# B&R Automation Studio project PLC code - cp (part 6)

#### HeightTracking.st
```iecst
ACTION RunHeightArray:

	// ------------------------------------------------------------------
	// Matrix advance and calculate the maximum

	//Move the values of the array
	ShiftArrayForward(ADR(iHeightArray), SIZEOF(iHeightArray), SIZEOF(iHeightArray[0]), iPositionsToRunArray, iTotalBlocksLengh);

	// High Ctrl data to Matrix
	// Loading data from sensors to
	IF gPhotoCells.status.xInstalled THEN
		LoadHeightFromArraySensor;
	END_IF
	IF gDing.State.xDingInstalled OR gBasicDetectMedia.Status.xInstalled THEN
		LoadHeightFromAnalogSensor;
	END_IF

	// Analyze height data and assign maximum height per section
	ResetMaxHeigh;
	FOR iIndexArray:= iTotalBlocksLengh TO iPositionsToRunArray BY -1 DO
		//Update te value of the thickness in the matrix
		AssignMaxHeighIndex;
	END_FOR

END_ACTION

ACTION ResetMaxHeigh:

	// It allows changes on height block correction when It changes Hand Printer
	FOR iIndexSection:=1 TO iTotalSections DO
		iMaxHeigh[iIndexSection]:=0;
	END_FOR

END_ACTION

ACTION AssignMaxHeighIndex:

	//Calculate the maximum of each section
	FOR iIndexSection:=1 TO iTotalSections DO
		//If the section is not enabled, do not calculate any Max
		IF dataHeigh.parameters.sections[iIndexSection].xEnabled THEN

			//If the Section does not correspond with the Index in Matrix, do not calculate Max
			IF iIndexArray > dataHeigh.parameters.sections[iIndexSection].iStart AND
				iIndexArray <= dataHeigh.parameters.sections[iIndexSection].iEnd 	 THEN

				iMaxHeigh[iIndexSection]:= MAX(iHeightArray[iIndexArray], iMaxHeigh[iIndexSection]);
			END_IF
		END_IF

	END_FOR

END_ACTION

ACTION AssignMaxHeight:

	//Calculate the maximum of each section
	FOR iIndexSection:=1 TO iTotalSections DO
		//If the section is not enabled, do not calculate any Max
		IF dataHeigh.parameters.sections[iIndexSection].xEnabled THEN
			FOR iIndexArray:= dataHeigh.parameters.sections[iIndexSection].iStart TO dataHeigh.parameters.sections[iIndexSection].iEnd DO
				iMaxHeigh[iIndexSection]:= MAX(iHeightArray[iIndexArray], iMaxHeigh[iIndexSection]);
			END_FOR
		END_IF
	END_FOR

END_ACTION

ACTION LoadHeightFromAnalogSensor:
	//TODO. convert in a FUNCTION to use 3 times

	// Fill-in moved spaces with new data
	iCurrentMediaHeight := 0;
	IF dataHeigh.Internal.iFastValues >= iPositionsToRunArray THEN
		// More values than holes to fill-in. Distribution of data
		rValuesPerPosition :=  dataHeigh.Internal.rFastValues / UINT_TO_REAL(iPositionsToRunArray);
		FOR iIndexArray:=0 TO iPositionsToRunArray -1 DO
			iHeightArray[iIndexArray + iAnalogSensorPosition] := 0;
			FOR iIndexNewMediaArray := INT_TO_UINT( TRUNC(UINT_TO_REAL(iIndexArray) * rValuesPerPosition )) TO INT_TO_UINT(TRUNC(UINT_TO_REAL(iIndexArray) * rValuesPerPosition )) DO
				iHeightArray[iIndexArray + iAnalogSensorPosition] := MAX(iHeightArray[iIndexArray + iAnalogSensorPosition], dataHeigh.Internal.AnalogHeightValues[iIndexNewMediaArray]);
				iCurrentMediaHeight := MAX(iCurrentMediaHeight, dataHeigh.Internal.AnalogHeightValues[iIndexNewMediaArray]);
			END_FOR
		END_FOR
	ELSE
		// More holes than data. Ampliation of data
		rValuesPerPosition :=  UINT_TO_REAL(iPositionsToRunArray) / dataHeigh.Internal.rFastValues;
		FOR iIndexNewMediaArray:=0 TO REAL_TO_UINT(dataHeigh.Internal.rFastValues) -1 DO
			FOR iIndexArray := INT_TO_UINT(TRUNC(UINT_TO_REAL(iIndexNewMediaArray) * rValuesPerPosition )) TO INT_TO_UINT(TRUNC(UINT_TO_REAL(iIndexNewMediaArray) * rValuesPerPosition )) DO
				iHeightArray[iIndexArray + iAnalogSensorPosition] :=dataHeigh.Internal.AnalogHeightValues[iIndexNewMediaArray];
				iCurrentMediaHeight := MAX(iCurrentMediaHeight, dataHeigh.Internal.AnalogHeightValues[iIndexNewMediaArray]);
			END_FOR
		END_FOR
	END_IF
	gThicknessCtrl.status.Heigh.iMediaHeigh := iCurrentMediaHeight;

END_ACTION

ACTION LoadHeightFromArraySensor:
	//TODO. convert in a FUNCTION to use 3 times

	// Fill-in moved spaces with new data
	iCurrentMediaHeight := 0;
	IF dataHeigh.Internal.iFastValues >= iPositionsToRunArray THEN
		// More values than holes to fill-in. Distribution of data
		rValuesPerPosition :=  dataHeigh.Internal.rFastValues / UINT_TO_REAL(iPositionsToRunArray);
		FOR iIndexArray:=0 TO iPositionsToRunArray -1 DO
			iHeightArray[iIndexArray + iArraySensorPosition] := 0;
			FOR iIndexNewMediaArray := INT_TO_UINT(TRUNC(UINT_TO_REAL(iIndexArray) * rValuesPerPosition )) TO INT_TO_UINT(TRUNC(UINT_TO_REAL(iIndexArray) * rValuesPerPosition )) DO
				iHeightArray[iIndexArray + iArraySensorPosition] := MAX(iHeightArray[iIndexArray + iArraySensorPosition], dataHeigh.Internal.ArrayHeightValues[iIndexNewMediaArray]);
				iCurrentMediaHeight := MAX(iCurrentMediaHeight, dataHeigh.Internal.ArrayHeightValues[iIndexNewMediaArray]);
			END_FOR
		END_FOR
	ELSE
		// More holes than data. Ampliation of data
		rValuesPerPosition :=  UINT_TO_REAL(iPositionsToRunArray) / dataHeigh.Internal.rFastValues;
		FOR iIndexNewMediaArray:=0 TO REAL_TO_UINT(dataHeigh.Internal.rFastValues) -1 DO
			FOR iIndexArray := INT_TO_UINT(TRUNC(UINT_TO_REAL(iIndexNewMediaArray) * rValuesPerPosition )) TO INT_TO_UINT(TRUNC(UINT_TO_REAL(iIndexNewMediaArray) * rValuesPerPosition )) DO
				iHeightArray[iIndexArray + iArraySensorPosition] :=dataHeigh.Internal.ArrayHeightValues[iIndexNewMediaArray];
				iCurrentMediaHeight := MAX(iCurrentMediaHeight, dataHeigh.Internal.ArrayHeightValues[iIndexNewMediaArray]);
			END_FOR
		END_FOR
	END_IF
	gThicknessCtrl.status.Heigh.iMediaHeigh := iCurrentMediaHeight;

END_ACTION
```

#### MediaTrackingFunct.st
```iecst
ACTION MoveMediaFromNewToInsideL1:

	IF MediaTracking_iTotalInsideL1 = THICK_MEDIATRACKING_MAX_MEDIA THEN
		// TODO: Raise alarm of received media without free space
		RETURN;
	END_IF

	// Moving from New to Inside
	IF dataHeigh.status.xNewMediaStackEnabled THEN
		// Managing Media and Energy
		MediaTrackingInsideL1[MediaTracking_iTotalInsideL1] := NewMediaStackL1[0];
	ELSE
		// Manage Energy information
		MediaEnergyRackL1[EnergyRack_iIndexL1] := dataHeigh.parameters.ContinuousMedia.Energy;
		MediaTrackingInsideL1[MediaTracking_iTotalInsideL1].iIndexMediaEnergy := EnergyRack_iIndexL1;
		MediaTrackingInsideL1[MediaTracking_iTotalInsideL1].pMediaEnery := ADR(MediaEnergyRackL1[EnergyRack_iIndexL1]);
		EnergyRack_iIndexL1 := EnergyRack_iIndexL1 + 1;
		IF EnergyRack_iIndexL1 > THICK_MEDIATRACKING_MAX_MEDIA_x2 THEN
			EnergyRack_iIndexL1 := 0;
		END_IF
		// Managing media
		MediaTrackingInsideL1[MediaTracking_iTotalInsideL1].Media := dataHeigh.parameters.ContinuousMedia.MediaData;
	END_IF

	MediaTrackingInsideL1[MediaTracking_iTotalInsideL1].HeadPosition := iIndexEnteringMedia;
	MediaTracking_iTotalInsideL1 := MediaTracking_iTotalInsideL1 + 1;
	AssignEnteringMediaL1;

	// Removing from New overwriting the array
	IF dataHeigh.status.xNewMediaStackEnabled THEN
		ShiftArrayBackward(ADR(NewMediaStackL1), SIZEOF(NewMediaStackL1), SIZEOF(NewMediaStackL1[0]), 1, Stack_iTotalNewMediaL1);
		Stack_iTotalNewMediaL1 := UINT_SUB(Stack_iTotalNewMediaL1, 1);
	END_IF

	AddMediaTrackingEvents(diTotalCmBelt, HEAD_DETECTED, ADR(TrackingEventsArray));

END_ACTION

ACTION MoveMediaFromNewToInsideL2:

	IF MediaTracking_iTotalInsideL2 = THICK_MEDIATRACKING_MAX_MEDIA THEN
		// TODO: Raise alarm of received media without free space
		RETURN;
	END_IF

	// Moving from New to Inside
	IF dataHeigh.status.xNewMediaStackEnabled THEN
		// Managing Media and Energy
		MediaTrackingInsideL2[MediaTracking_iTotalInsideL2] := NewMediaStackL2[0];
	ELSE
		// Manage Energy information
		MediaEnergyRackL2[EnergyRack_iIndexL2] := dataHeigh.parameters.ContinuousMedia.Energy;
		MediaTrackingInsideL2[MediaTracking_iTotalInsideL2].iIndexMediaEnergy := EnergyRack_iIndexL2;
		MediaTrackingInsideL2[MediaTracking_iTotalInsideL2].pMediaEnery := ADR(MediaEnergyRackL2[EnergyRack_iIndexL2]);
		EnergyRack_iIndexL2 := EnergyRack_iIndexL2 + 1;
		IF EnergyRack_iIndexL2 > THICK_MEDIATRACKING_MAX_MEDIA_x2 THEN
			EnergyRack_iIndexL2 := 0;
		END_IF
		// Managing media
		MediaTrackingInsideL2[MediaTracking_iTotalInsideL2].Media := dataHeigh.parameters.ContinuousMedia.MediaData;
	END_IF

	MediaTrackingInsideL2[MediaTracking_iTotalInsideL2].HeadPosition := iIndexEnteringMedia;
	MediaTracking_iTotalInsideL2 := MediaTracking_iTotalInsideL2 + 1;
	AssignEnteringMediaL2;

	// Removing from New overwriting the array
	IF dataHeigh.status.xNewMediaStackEnabled THEN
		ShiftArrayBackward(ADR(NewMediaStackL2), SIZEOF(NewMediaStackL2), SIZEOF(NewMediaStackL2[0]), 1, Stack_iTotalNewMediaL2);
		Stack_iTotalNewMediaL2 := UINT_SUB(Stack_iTotalNewMediaL2, 1);
	END_IF

	AddMediaTrackingEvents(diTotalCmBelt, HEAD_DETECTED, ADR(TrackingEventsArray));

END_ACTION

ACTION MoveMediaFromInsideToOutL1:

	// Removing from New overwriting the array
	ShiftArrayBackward(ADR(MediaTrackingInsideL1), SIZEOF(MediaTrackingInsideL1), SIZEOF(MediaTrackingInsideL1[0]), 1, MediaTracking_iTotalInsideL1);
	MediaTracking_iTotalInsideL1 := UINT_SUB(MediaTracking_iTotalInsideL1, 1);
	AssignEnteringMediaL1;
	xExitingMediaL1 := TRUE;

END_ACTION

ACTION MoveMediaFromInsideToOutL2:

	// Removing from New overwriting the array
	ShiftArrayBackward(ADR(MediaTrackingInsideL2), SIZEOF(MediaTrackingInsideL2), SIZEOF(MediaTrackingInsideL2[0]), 1, MediaTracking_iTotalInsideL2);
	MediaTracking_iTotalInsideL2 := UINT_SUB(MediaTracking_iTotalInsideL2, 1);
	AssignEnteringMediaL2;
	xExitingMediaL2 := TRUE;

END_ACTION

ACTION AssignEnteringMediaL1:

	// Need to protect the case when exiting one media and no other media inside. In this case pointing to an empty location, but no errors
	IF MediaTracking_iTotalInsideL1 > 0 THEN
		EnteringMediaL1 ACCESS ADR(MediaTrackingInsideL1[MediaTracking_iTotalInsideL1-1].Media);
	ELSE
		EnteringMediaL1 ACCESS ADR(MediaTrackingInsideL1[0].Media);
	END_IF

END_ACTION

ACTION AssignEnteringMediaL2:

	// Need to protect the case when exiting one media and no other media inside. In this case pointing to an empty location, but no errors
	IF MediaTracking_iTotalInsideL2 > 0 THEN
		EnteringMediaL2 ACCESS ADR(MediaTrackingInsideL2[MediaTracking_iTotalInsideL2-1].Media);
	ELSE
		EnteringMediaL2 ACCESS ADR(MediaTrackingInsideL2[0].Media);
	END_IF

END_ACTION

ACTION RunMediaInsidePositions:

	RunMediaInsidePositionsL1;
	IF dataHeigh.parameters.xDoubleLine THEN
		RunMediaInsidePositionsL2;
	END_IF

END_ACTION

ACTION RunMediaInsidePositionsL1:

	IF MediaTracking_iTotalInsideL1 = 0 THEN
		RETURN;
	END_IF

	FOR iIndexArray := 0 TO MediaTracking_iTotalInsideL1 -1 DO
		MediaTrackingInsideL1[iIndexArray].HeadPosition := MediaTrackingInsideL1[iIndexArray].HeadPosition + iPositionsToRunArray;
		// If tail position is <>0 is because it has been asigned
		IF MediaTrackingInsideL1[iIndexArray].TailPosition <> 0 THEN
			MediaTrackingInsideL1[iIndexArray].TailPosition := MediaTrackingInsideL1[iIndexArray].TailPosition + iPositionsToRunArray;
		END_IF
	END_FOR

END_ACTION

ACTION RunMediaInsidePositionsL2:

	IF MediaTracking_iTotalInsideL2 = 0 THEN
		RETURN;
	END_IF

	FOR iIndexArray := 0 TO MediaTracking_iTotalInsideL2 -1 DO
		MediaTrackingInsideL2[iIndexArray].HeadPosition := MediaTrackingInsideL2[iIndexArray].HeadPosition + iPositionsToRunArray;
		// If tail position is <>0 is because it has been asigned
		IF MediaTrackingInsideL2[iIndexArray].TailPosition <> 0 THEN
			MediaTrackingInsideL2[iIndexArray].TailPosition := MediaTrackingInsideL2[iIndexArray].TailPosition + iPositionsToRunArray;
		END_IF
	END_FOR

END_ACTION
```

#### RejectTracking.st
```iecst
ACTION RunRejectArray:

	//Need to run the matrix through all belts
	ShiftArrayForward(ADR(ValidMedia), SIZEOF(ValidMedia), SIZEOF(ValidMedia[0]), iPositionsToRunArray, iMaxTrackingPosition + 5);

	// To Clarify if Command for 1 or Order for all till contrary order
	IF EDGEPOS(dataHeigh.Commands.xRushProof) THEN
		xRushProof:=TRUE;
		iRushProofCounter := iRushProofCounter + 1; //To be shown on UI. Useful for users and debugging
		LogRushProof;

		MarkBoardAsRejectedToTheFrontEdge;
	END_IF

	// When receiving the signal of media detected to Reject, run the matrix and mark all boards as ToReject
	// This will ocurr the next scan cycle of the detection, but it is no a problem in this case
	IF EDGENEG(dataHeigh.parameters.xBlockInProperPrintingPosition) OR dataHeigh.status.Detection.xMediaToRejectDetected THEN
		IF gMachine.St.AutoMode.xProduction THEN
			MarkAllBoardsBelowMachineAsRejected;
		END_IF
		xReturningFromReject := TRUE;
	END_IF

	//To write the matrix
	IF dataHeigh.parameters.xBlockInProperPrintingPosition AND NOT dataHeigh.Orders.xDiscardAllMedia THEN
		IF NOT xRushProof THEN

			IF NOT xReturningFromReject THEN
				// This is the standard behaviour. MOST OF TIMES THROUGH HERE
				iNewValidMedia := MEDIATRACKING_VALID;
				LoadNewValidMediaData;
			ELSE
				//   This is the behaviourr while finishing the Reject state,
				// and searching for a gap in the media entering to considering finished
				IF dataHeigh.parameters.Detection.ProductDetect.xFixedSensor THEN
					iNewValidMedia := MEDIATRACKING_INVALID;
				ELSE
					iNewValidMedia := MEDIATRACKING_UNKNOWN;
				END_IF
				LoadNewValidMediaData;
				DetectGapEnteringTheMachine;
			END_IF
		ELSE
			// Review Rear Edge. Invalid if not Edge. Valid after the edge
			CheckRearEdgeofRejectedBoard;
		END_IF
	ELSE
		IF dataHeigh.parameters.Detection.ProductDetect.xFixedSensor THEN
			iNewValidMedia := MEDIATRACKING_INVALID;
		ELSE
			iNewValidMedia := MEDIATRACKING_UNKNOWN;
		END_IF
		LoadNewValidMediaData;

		xRushProof:=FALSE;
	END_IF

	// Just update if the new data is written in the positions moved previously

END_ACTION

ACTION LoadNewValidMediaData:
	FOR iIndexArray := 0 TO iPositionsToRunArray -1 DO
		ValidMedia[iIndexArray + iProductDetectSensorPosition] := iNewValidMedia;
	END_FOR
END_ACTION

ACTION ReviewRejectActivation:

	//[RGP] This part must be located in code executed much faster: less than (MinGap/MaxBeltSpeed)
	//We need TO force gaps TO be written with a PDsignal filter, TO avoid "iPositionsToRunArray" TO mask them
	//we can check previous index (iRejectLengthAdjustment-X). X: Positions in matrix forced to be 0, as a gap

	FastReviewReject;

	//Overwritting valid media array to mark boards below bars when block raises to safe position
	//[RGP] 15274: Overwritting matrix position to know which boards are below block's bars when empty belt mode.
	IF EDGEPOS(dataHeigh.Orders.xDiscardAllMedia) THEN
		FOR iIndex := dataHeigh.parameters.Detection.ProductDetect.iSensorPosition TO dataHeigh.parameters.iTotalBlocksLengh DO
			IF dataHeigh.parameters.Detection.ProductDetect.xFixedSensor THEN
				ValidMedia[iIndex] := MEDIATRACKING_INVALID;
			ELSE
				ValidMedia[iIndex] := MEDIATRACKING_UNKNOWN;
			END_IF
		END_FOR
	END_IF

	ton_PhysicalHoldReject(IN:=gMachine.In.Buttons.xReset, PT:=T#2S);
	xHoldReject := ValidMedia[iHoldRejectLengthAdjustment] = MEDIATRACKING_UNKNOWN;

	IF EDGEPOS(xHoldReject) THEN
		AddMediaTrackingEvents(diTotalCmBelt + iHoldRejectLengthAdjustment, START_HOLDREJEC, ADR(TrackingEventsArray));
	END_IF
	IF EDGENEG(xHoldReject) THEN
		AddMediaTrackingEvents(diTotalCmBelt + iHoldRejectLengthAdjustment, END_HOLDREJECT, ADR(TrackingEventsArray));
	END_IF

	// Out signals
	dataHeigh.Outputs.xHoldReject := ton_PhysicalHoldReject.Q OR xHoldReject;

END_ACTION

ACTION MarkBoardAsRejectedToTheFrontEdge:

	// Searching for the gap in xMediaTracking
	FOR iIndex:=iProductDetectSensorPosition TO iMAXTRACKINGARRAY DO
		// Searching for the gap in xMediaTracking to Stop
		IF xMediaTracking[iIndex] = 0  THEN
			EXIT;
		END_IF
		ValidMedia[iIndex] := MEDIATRACKING_INVALID;
	END_FOR

END_ACTION

ACTION DetectGapEnteringTheMachine:

	// Searching for the gap in xMediaTracking
	FOR iIndex:=iProductDetectSensorPosition + iPositionsToRunArray TO iProductDetectSensorPosition BY -1 DO
		// Searching for the gap in xMediaTracking to Stop
		IF xMediaTracking[iIndex] = 0  THEN
			xReturningFromReject := FALSE;
			EXIT;
		END_IF
	END_FOR

END_ACTION

ACTION CheckRearEdgeofRejectedBoard:

	// Searching for the gap in xMediaTracking
	FOR iIndex:=iProductDetectSensorPosition + iPositionsToRunArray TO iProductDetectSensorPosition BY -1 DO

		IF xMediaTracking[iIndex] = 0  AND xRushProof THEN
			// Detected the Rear Edge of the board. Now not in RushProof
			ValidMedia[iIndex] := MEDIATRACKING_INVALID;
			xRushProof:=FALSE;
		ELSIF NOT xRushProof THEN
			ValidMedia[iIndex] := MEDIATRACKING_VALID;
		ELSE
			ValidMedia[iIndex] := MEDIATRACKING_INVALID;
		END_IF

	END_FOR

END_ACTION

ACTION MarkAllBoardsBelowMachineAsRejected:

	// Marking all positions below machine as Invalid
	xMarkLastBoardBelowBlock := TRUE; //To avoid mark a board half unknown - half invalid, in case of using full stacker is not sent using reject sheet, and the holdreject signal is sent too late
	FOR iIndex := dataHeigh.parameters.Detection.ProductDetect.iSensorPosition + iPositionsToRunArray TO dataHeigh.parameters.iTotalBlocksLengh DO
		IF xMediaTracking[iIndex] = 1 AND xMarkLastBoardBelowBlock THEN
			IF dataHeigh.parameters.Detection.ProductDetect.xFixedSensor THEN
				ValidMedia[iIndex] := MEDIATRACKING_INVALID;
			ELSE
				ValidMedia[iIndex] := MEDIATRACKING_UNKNOWN;
			END_IF
		ELSE
			xMarkLastBoardBelowBlock := FALSE;
			IF ValidMedia[iIndex] <> MEDIATRACKING_UNKNOWN THEN
				ValidMedia[iIndex] := MEDIATRACKING_INVALID;
			END_IF
		END_IF
	END_FOR

	//  If there is a board inside the machine, but with the head outside the machine,
	// mark all that board as ToReject. The rear side won't be properly printed
	FOR iIndex:=dataHeigh.parameters.iTotalBlocksLengh TO iMAXTRACKINGARRAY DO
		// Searching for the gap in xMediaTracking to Stop
		IF xMediaTracking[iIndex] = 0 THEN
			EXIT;
		END_IF
		IF ValidMedia[iIndex] <> MEDIATRACKING_UNKNOWN THEN
			ValidMedia[iIndex] := MEDIATRACKING_INVALID;
		END_IF
	END_FOR

END_ACTION
```

#### AlarmsCheckMedia.st
```iecst
ACTION AlarmsCheckMedia:

	FilterCheckMediaInputs;

	FOR iIndexCheck:=1 TO 1 DO
	//FOR iIndexCheck:=1 TO MAX_LAST_CHECKMEDIA DO
		CheckMediaIndex;
	END_FOR

	IF EDGEPOS(dataHeigh.Inputs.CheckMedia[1].xCheckFail) THEN
		iTotalCheckMediaBoards := iTotalCheckMediaBoards +1;
	END_IF

END_ACTION

ACTION CheckMediaIndex:

	IF NOT dataHeigh.parameters.CheckMedia[iIndexCheck].xActive THEN
		RETURN;
	END_IF

	CheckMediaWork ACCESS ADR(dataHeigh.parameters.CheckMedia[iIndexCheck]);

	CheckMediaFrontEdgeBoardSearch;

	IF xFrontEdgeBoardInChekMedia AND NOT tofNewCheckBoardTracking.Q THEN
		iTotalCheckMediaTrackingBoards := iTotalCheckMediaTrackingBoards + 1;
	END_IF
	tofNewCheckBoardTracking.IN := xFrontEdgeBoardInChekMedia;
	tofNewCheckBoardTracking.PT := t#500ms;
	tofNewCheckBoardTracking();

	IF xFrontEdgeBoardInChekMedia AND NOT dataHeigh.Internal.CheckMediaFilteredSensors[1] THEN
		dataHeigh.Alarms.CheckMediaHead[iIndexCheck] := TRUE;
	END_IF

	IF CheckMediaWork.xCheckGap THEN
		CheckMediaTailEdgeBoardSearch;
		IF xRearEdgeBoardInChekMedia AND dataHeigh.Internal.CheckMediaFilteredSensors[1] THEN
			dataHeigh.Alarms.CheckMediaTail[iIndexCheck] := TRUE;
		END_IF
	END_IF

	// Assigning the summary alarm
	IF dataHeigh.Alarms.CheckMediaHead[iIndexCheck] OR dataHeigh.Alarms.CheckMediaTail[iIndexCheck] THEN
		dataHeigh.Alarms.CheckMedia[iIndexCheck] := TRUE;
	END_IF

END_ACTION

ACTION CheckMediaFrontEdgeBoardSearch:

	iIndexPositionToReviewMedia:= CheckMediaWork.CheckPosition + CheckMediaWork.CheckDelayPosition - MAX(1, iPositionsToRunArray + 2); //Increasing the quantity of data to avoid not checking any position during accelerations

	xFrontEdgeBoardInChekMedia := FALSE;
	// Search for the boards "head" in Sensor position
	FOR iIndexMediaPresent := CheckMediaWork.CheckPosition + CheckMediaWork.CheckDelayPosition TO iIndexPositionToReviewMedia BY -1 DO
		IF xMediaTracking[iIndexMediaPresent] > 0 AND xMediaTracking[iIndexMediaPresent+1] = 0 THEN
			xFrontEdgeBoardInChekMedia:=TRUE;
		END_IF
	END_FOR

END_ACTION

ACTION CheckMediaTailEdgeBoardSearch:

	iIndexPositionToReviewMedia:= CheckMediaWork.CheckPosition + CheckMediaWork.CheckDelayPosition - MAX(1, iPositionsToRunArray + 2); //Increasing the quantity of data to avoid not checking any position during accelerations

	xRearEdgeBoardInChekMedia := FALSE;
	// Search for the boards "head" in Sensor position
	FOR iIndexMediaPresent := CheckMediaWork.CheckPosition + CheckMediaWork.CheckDelayPosition TO iIndexPositionToReviewMedia BY -1 DO
		IF xMediaTracking[iIndexMediaPresent] = 0 AND xMediaTracking[iIndexMediaPresent+1] > 0 THEN
			xRearEdgeBoardInChekMedia:=TRUE;
		END_IF
	END_FOR

END_ACTION

// This action is called before checking the alarms
ACTION FilterCheckMediaInputs:

	tonFilterCheckMediaSensor[1].IN := NOT EDGE(dataHeigh.Inputs.CheckMedia[1].xCheckFail);
	tonFilterCheckMediaSensor[1].PT := TimeFromMmAndMmin(dataHeigh.parameters.CheckMedia[1].iSensorFilter, dataHeigh.parameters.Belt.rBeltSpeed) ;
	tonFilterCheckMediaSensor[1]();

	// Just with the signal stable raises the timer
	IF EDGEPOS(tonFilterCheckMediaSensor[1].Q) THEN
		dataHeigh.Internal.CheckMediaFilteredSensors[1] := dataHeigh.Inputs.CheckMedia[1].xCheckFail;
		IF dataHeigh.Inputs.CheckMedia[1].xCheckFail THEN
			iTotalCheckMediaTrackBoardsFilt := iTotalCheckMediaTrackBoardsFilt + 1;
		END_IF
	END_IF

END_ACTION
```

#### AlarmsSummary.st - Alarms summary
```iecst
ACTION AlarmsSummary:

	//Alarms STOP
	iReasonStop.0 := dataHeigh.Alarms.CheckMedia[1];
	iReasonStop.1 := dataHeigh.Alarms.CheckMedia[2];

	dataHeigh.AlSummary.xAlarmStop := iReasonStop > 0;
	IF EDGEPOS(dataHeigh.AlSummary.xAlarmStop) THEN
		dataHeigh.AlSummary.iReasonStop[0] := iReasonStop;
	ELSIF EDGEPOS(NOT dataHeigh.parameters.AutoMode.xStop AND NOT dataHeigh.AlSummary.xAlarmStop) THEN
		dataHeigh.AlSummary.iReasonStop[0] := 0;
	END_IF

	//Alarms CRITICAL
	iReasonCritical.0 := FALSE;

	dataHeigh.AlSummary.xAlarmCritical := iReasonCritical > 0;
	IF dataHeigh.parameters.Mode.xAuto AND EDGEPOS(dataHeigh.AlSummary.xAlarmCritical) THEN
		dataHeigh.AlSummary.iReasonCritical := iReasonCritical;
	ELSIF EDGEPOS(dataHeigh.parameters.Mode.xAuto AND NOT dataHeigh.AlSummary.xAlarmCritical) THEN
		dataHeigh.AlSummary.iReasonCritical := 0;
	END_IF

END_ACTION
```

#### EventLog.st
```iecst
ACTION LogRejectingEnded:
	stEventLogEndRejecting.Source := ELOG_TYPE_DETECTION;
	stEventLogEndRejecting.Severity:= ELOG_SEVERITY_INFO;
	stEventLogEndRejecting.Facility:= 0;
	stEventLogEndRejecting.ErrorCode:=0;
	stEventLogEndRejecting.Text := 'ThickCtrl. End Rejected Media Inside';
	gEventLogLoader(EventData := ADR(stEventLogEndRejecting));
END_ACTION

ACTION LogRushProof:
	stEventLogRushProof.Source := ELOG_TYPE_DETECTION;
	stEventLogRushProof.Severity:= ELOG_SEVERITY_INFO;
	stEventLogRushProof.Facility:= 0;
	stEventLogRushProof.ErrorCode:=0;
	stEventLogRushProof.Text := 'gThicknessCtrl.Commands.xRushProof received. Rush proof counter: ';
	// Adding counter number to log message
	brsitoa(iRushProofCounter, ADR(strAuxEventDesc));
	brsstrcat(ADR(stEventLogRushProof.Text), ADR(strAuxEventDesc));

	gEventLogLoader(EventData := ADR(stEventLogRushProof));
END_ACTION
```

#### ThicknessCtrl.var
```iecst
VAR
	iMediaHeight : UINT;
	dataHeigh : REFERENCE TO stThicknessCtrl_typ;
	RTInfo_0 : RTInfo;
	rPeriode : REAL := 0; (*Cycle time in microseconds. Read just in INIT. NEVER Write over it!!!*)
	iIndexArray : UINT;
	iIndexNewMediaArray : UINT;
	iIndexEnteringMedia : UINT;
	iIndexFinishEnteringMedia : UINT;
	iIndexExitingMedia : UINT;
	rAccumAdvBelt : REAL;
	iMediaFilter : UINT; (*Cm to consider that pd signal has detected a board*)
	iIndexCuringTrackingMatrix : UINT;
	xCuringTracking : ARRAY[0..iMAXTRACKINGARRAY] OF USINT; (*Matrix with the information about media that need to be cured. Each position corresponds to a cm. Bit 0: L1 Color, Bit 1 L1 White, Bit 2 L2 Color, Bit 3 L2 White*)
	ValidMedia : ARRAY[0..iMAXTRACKINGARRAY] OF SINT; (*Array with the information about valid media. -1 means no information about media so HoldReject, 0 means invalid media, 1 means valid media. Each position corresponds to a cm*)
	xMediaTracking : ARRAY[0..iMAXTRACKINGARRAY] OF USINT; (*Matrix with the information about if there is Media in the position. Each position corresponds to a cm. Bit 0: L1 , Bit 1 L2*)
	xMediaPresentAnalog : ARRAY[0..iMAXMEDIAPRESENTARRAY] OF BOOL; (*Matrix with the information about if there is Media detected from the ARRAY sensor in the position. Each position corresponds to a cm*)
	xMediaPresentArray : ARRAY[0..iMAXMEDIAPRESENTARRAY] OF BOOL; (*Matrix with the information about if there is Media detected from the ARRAY sensor in the position. Each position corresponds to a cm*)
	xMediaPresentBasic : ARRAY[0..iMAXMEDIAPRESENTARRAY] OF BOOL; (*Matrix with the information about if there is Media detected from the ARRAY sensor in the position. Each position corresponds to a cm*)
	iHeightArray : ARRAY[0..iMAXHEIGHTARRAY] OF UINT;
	iDistanceBeltTurn : UINT; (*Distance to know when a belt cycle has been run*)
	iDistanceWorkEmptyBelt : UINT;
	iDistanceMountPieceOut : UINT;
	iDistanceMediaInside : UINT;
	iDistanceVirtualMediaInside : UINT;
	iDistanceMediaToRejectInside : UINT;
	iDistanceTrackingEmpty : UINT;
	iIndexSection : USINT;
	iIndexCheck : USINT;
	CheckMediaWork : REFERENCE TO stThicknessCtrl_CheckMediaParams; (*Variable inside the FOR to work with*)
	iLastMaxHeigh : ARRAY[0..TOTAL_THICKNESS_SECTIONS] OF UINT;
	iMaxHeigh : ARRAY[0..TOTAL_THICKNESS_SECTIONS] OF UINT;
	iCountIncrease : ARRAY[0..TOTAL_THICKNESS_SECTIONS] OF UINT;
	iTotalBlocksLengh : UINT; (*Value in cm. Max is 600*)
END_VAR
VAR CONSTANT
	MM_PERPOSITION_IN_ARRAY : REAL := 10.0;
END_VAR
VAR
	iTotalSections : USINT; (*Sections configured in the machine*)
	rMinBeltSpeedToStart : REAL;
	iPositionsToRunArray : UINT;
	iRushProofCounter : INT;
	tonResetRushProofCounterTimer : TON;
	xResetRejectRushProofCounter : BOOL;
	xRushProof : BOOL;
	xCameraRejectSignal : BOOL;
	xReject : BOOL;
	xReviewRejectOrder : BOOL;
	xHoldReject : BOOL;
	tp_Reject : TP;
	tp_RejectLongTime : TP;
	ton_PhysicalHoldReject : TON;
	iProductDetectSensorPosition : UINT; (*Position of the sensor in X direction in cm*)
	iArraySensorPosition : INT; (*Position of the sensor in X direction in cm*)
	iAnalogSensorPosition : INT; (*Position of the sensor in X direction in cm*)
	iDetectionMediaSensorPosition : INT;
	iLastPosition : INT;
	iHoldRejectLengthAdjustment : UINT;
	iRejectLengthAdjustment : UINT;
	iMaxTrackingPosition : UINT;
	iIndex : UINT;
	iStartCuringWindow : INT; (*Distance in cm*)
	iEndCuringWindow : INT; (*Distance in cm*)
	iIndexWindow : UINT;
	iReasonMediaBelow : USINT;
	iIndexPositionToReviewMedia : UINT;
	iBoardsBelowBlockL1 : UINT;
	iBoardsBelowBlockL2 : UINT;
	iIndexMediaPresent : UINT;
	rValuesPerPosition : REAL;
	iNumberOfPositionsToBeUpdated : UINT; (*Matrix's number of positions to update*)
	xFilteredProductDetectMediaL1 : BOOL;
	xFilteredProductDetectMediaL2 : BOOL;
	xFilteredAnalogSensorMedia : BOOL;
	xFilteredArraySensorMedia : BOOL;
	xFilteredBasicDetectionMedia : BOOL;
	iNewValidMedia : SINT;
	iCurrentMediaHeight : UINT;
	xFrontEdgeBoardInChekMedia : BOOL;
	xRearEdgeBoardInChekMedia : BOOL;
	ars_CheckMedia : ARRAY[0..MAX_LAST_CHECKMEDIA] OF AutoResetSound;
	ars_NoThicknessSystemInstalled : AutoResetSound;
	iReasonSound : UINT;
	stAlarmsReseted : stThicknessCtrl_Alarms_typ;
	stAlarmsSummaryReseted : stEFI_AlarmSummary;
	iReasonStop : UINT;
	iReasonCritical : UINT;
	xMountedMedia : BOOL; (*Previously as an input, now ThicknessCtrl reads the value from AnalogCtrl and ArrayCtrl*)
	LoadNewMedia_MethodOperate : UaSrv_MethodOperate;
	LoadNewMedia_Step : USINT;
	LoadNewMedia_Media : stThicknessCtrl_MediaConfig;
	LoadNewMedia_Result : UDINT;
	LoadNewMedia_ErrorID : UDINT;
	LoadNewMedia_ReviewResult : UDINT;
	InsertNewMedia_MethodOperate : UaSrv_MethodOperate;
	InsertNewMedia_Step : USINT;
	InsertNewMedia_Id : DINT;
	InsertNewMedia_Media : stThicknessCtrl_MediaConfig;
	InsertNewMedia_Result : UDINT;
	InsertNewMedia_ErrorID : UDINT;
	InsertNewMedia_ReviewResult : UDINT;
	InsertNewMedia_Position : UINT;
	RemoveNewMedia_MethodOperate : UaSrv_MethodOperate;
	RemoveNewMedia_Step : USINT;
	RemoveNewMedia_Line : USINT;
	RemoveNewMedia_Id : DINT;
	RemoveNewMedia_Result : UDINT;
	RemoveNewMedia_ErrorID : UDINT;
	RemoveNewMedia_ReviewResult : UDINT;
	RemoveNewMedia_Position : UINT;
	LoadNewMediaEnergy_MethodOperate : UaSrv_MethodOperate;
	LoadNewMediaEnergy_Step : USINT;
	LoadNewMediaEnergy_Media : stThickCtrl_EnergyMedia;
	LoadNewMediaEnergy_Result : UDINT;
	LoadNewMediaEnergy_ErrorID : UDINT;
	LoadNewMediaEnergy_ReviewResult : UDINT;
	LoadNewMediaEnergy_Position : UINT;
	InsertNewMediaEn_MethodOperate : UaSrv_MethodOperate;
	InsertNewMediaEn_Step : USINT;
	InsertNewMediaEn_Id : DINT;
	InsertNewMediaEn_Media : stThickCtrl_EnergyMedia;
	InsertNewMediaEn_Result : UDINT;
	InsertNewMediaEn_ErrorID : UDINT;
	InsertNewMediaEn_ReviewResult : UDINT;
	InsertNewMediaEn_Position : UINT;
	LoadNewMediaEnergyCont_MethodOp : UaSrv_MethodOperate;
	LoadNewMediaEnergyCont_Step : USINT;
	LoadNewMediaEnergyCont_Media : stThickCtrl_EnergyMedia;
	LoadNewMediaEnergyCont_Result : UDINT;
	LoadNewMediaEnergyCont_ErrorID : UDINT;
	LoadNewMediaEnergyCont_ReviewRes : UDINT;
	iIndexCleanMediaArray : UINT;
	iProdDetectFilterStartIndex : UINT;
	iSensorFilterStartIndex : UINT;
	iPositionAdjusted : UINT;
	NewMediaStackL1 : ARRAY[0..THICK_MEDIATRACKING_MAX_MEDIA] OF stThicknessCtrl_MediaPosStatus; (*FIFO Stack. Elements enter at the end, and go to First while exiting elements*)
	NewMediaStackL2 : ARRAY[0..THICK_MEDIATRACKING_MAX_MEDIA] OF stThicknessCtrl_MediaPosStatus; (*FIFO Stack. Elements enter at the end, and go to First while exiting elements*)
	MediaTrackingInsideL1 : REFERENCE TO ARRAY[0..THICK_MEDIATRACKING_MAX_MEDIA] OF stThicknessCtrl_MediaPosStatus; (*FIFO. Elements enter at the end, and go to First while exiting elements*)
	MediaTrackingInsideL2 : REFERENCE TO ARRAY[0..THICK_MEDIATRACKING_MAX_MEDIA] OF stThicknessCtrl_MediaPosStatus; (*FIFO. Elements enter at the end, and go to First while exiting elements*)
	MediaEnergyRackL1 : ARRAY[0..THICK_MEDIATRACKING_MAX_MEDIA_x2] OF stThickCtrl_Energy; (*Need the memory area for NewMedia and for MediaInside with full data*)
	MediaEnergyRackL2 : ARRAY[0..THICK_MEDIATRACKING_MAX_MEDIA_x2] OF stThickCtrl_Energy; (*Need the memory area for NewMedia and for MediaInside with full data*)
	Stack_iTotalNewMediaL1 : UINT;
	Stack_iTotalNewMediaL2 : UINT;
	MediaTracking_iTotalInsideL1 : UINT;
	MediaTracking_iTotalInsideL2 : UINT;
	MediaTracking_iTotalInsideL1_cp : UINT;
	MediaTracking_iTotalInsideL2_cp : UINT;
	MediaTracking_xEnteringMachineL1 : BOOL;
	MediaTracking_xEnteringMachineL2 : BOOL;
	EnergyRack_iIndexL1 : USINT; (*Index of the next free rack in array*)
	EnergyRack_iIndexL2 : USINT; (*Index of the next free rack in array*)
	xDetectedGap_L1 : BOOL;
	xDetectedGap_L2 : BOOL;
	EnteringMediaL1 : REFERENCE TO stThicknessCtrl_MediaPosStatus; (*Current media entering in the machine*)
	EnteringMediaL2 : REFERENCE TO stThicknessCtrl_MediaPosStatus; (*Current media entering in the machine*)
	EnteringMediaContinuous : stThicknessCtrl_MediaPosStatus; (*Current media entering in the machine*)
	xMediaInLedPositionWhiteL1 : BOOL;
	xMediaInLedPositionWhiteL2 : BOOL;
	xMediaInLedPositionPrimerL1 : BOOL;
	xMediaInLedPositionPrimerL2 : BOOL;
	xMediaInLedPositionColorL1 : BOOL;
	xMediaInLedPositionColorL2 : BOOL;
	CureLampParams : REFERENCE TO stThicknessCtrl_CureLampParams;
	CommandsReseted : stThicknessCtrl_Commands_typ;
	iSafetyMarginToHeight : UINT;
	xAddedSafetyMarginToHeight : BOOL;
	iIndexReviewArray : UINT;
	iFirstIndex : UINT;
	iLastIndex : UINT;
	xDetectionSystemIncoherenceL1 : BOOL; (*There is no media detection consistensy between PD an the array sensor . L1*)
	xDetectionSystemIncoherenceL2 : BOOL; (*There is no media detection consistensy between PD an the array sensor . L2*)
	EnergyTest : stThickCtrl_EnergyMedia;
	iIndexDryer : USINT;
	DryerInfo : REFERENCE TO stThicknessCtrl_NirDryerParams;
	iDistanceDelay : UINT; (*Distance in cm*)
	iDistanceWindow : UINT; (*Distance in cm*)
	MaxLampIntensityL1 : ARRAY[0..THICKENERGY_MAX_LAMPS] OF INT;
	MaxLampIntensityL2 : ARRAY[0..THICKENERGY_MAX_LAMPS] OF INT;
	LampIntensityL2 : ARRAY[0..THICKENERGY_MAX_LAMPS] OF INT;
	xReturningFromReject : BOOL;
	rMediaThicknessMargin : REAL;
	rMediaThickness : REAL;
	rSubstratePowerReduction : REAL; (*Iternal variable for Substrate power reduction. From 1.0 (default) to 0.3 is allowed*)
	rThermalInerciaReduction : REAL;
	rPowerReduction : REAL; (*Iternal variable for power reduction. Joining all power reductions*)
	diTotalCmBelt : UDINT;
	TrackingEventsArray : ARRAY[0..THICK_MAX_TRACKING_EVENTS] OF stThicknessCtrl_TrackingEvent;
	GetTOD : DTStructureGetTime;
	tiTimeOfDay : DTStructure;
	stEventLogEndRejecting : EventLog_typ;
	stEventLogResetRushProofCounter : EventLog_typ;
	stEventLogRushProof : EventLog_typ;
	strAuxEventDesc : STRING[129];
	iTotalCheckMediaTrackingBoards : UINT;
	iTotalCheckMediaTrackBoardsFilt : UINT;
	iTotalCheckMediaBoards : UINT;
	tofNewCheckBoardTracking : TOF;
	tonFilterCheckMediaSensor : ARRAY[0..MAX_LAST_CHECKMEDIA] OF TON;
	ExternalMediaConfig : REFERENCE TO stThicknessCtrl_MediaConfig;
	xExitingMediaL1 : BOOL;
	xExitingMediaL2 : BOOL;
	iForcedMovedOutMediaL1 : UDINT;
	iForcedMovedOutMediaL2 : UDINT;
	xMarkLastBoardBelowBlock : BOOL; (*TRUE when the ValidMedia values of the board below PD is set to UNKNOWN when marking all boards below machine as rejected*)
END_VAR
```

- TrackingStack.uam (not shown)

### Program Logical/ExtPack/_Media/ThicknessCtrl/ThicknessCtrl_v2/ThicknessCtrl_Fast (IEC)

#### ThickCtrl_Fast.st - Thickness Manager program
```iecst
PROGRAM _INIT

	RTInfo_0(enable :=TRUE );
	rPeriode:= UDINT_TO_REAL (RTInfo_0.cycle_time)/1000;  // Cycle time in microseconds
	gThicknessCtrl.Internal.rCycleFast := rPeriode;

END_PROGRAM

PROGRAM _CYCLIC

	IF gDing.State.xDingInstalled THEN

		ShiftArrayForward(ADR(gThicknessCtrl.Internal.AnalogHeightValues), SIZEOF(gThicknessCtrl.Internal.AnalogHeightValues), SIZEOF(gThicknessCtrl.Internal.AnalogHeightValues[0]), 1, THICK_MAX_UPDATE_VALUES);

		// Ding laser position to heigh detection ctrl
		gThicknessCtrl.Internal.AnalogHeightValues[0] := REAL_TO_UINT(MAX(gDing.State.rBarsPosition,
																		gThicknessCtrl.status.Heigh.rMediaThicknessMargin)*100);

		//Load array of data to avoid loosing information -----------------------------------------
		//Move the array one position
		ShiftArrayForward(ADR(gThicknessCtrl.Internal.MediaAnalogValues), SIZEOF(gThicknessCtrl.Internal.MediaAnalogValues), SIZEOF(gThicknessCtrl.Internal.MediaAnalogValues[0]), 1, THICK_MAX_UPDATE_VALUES);
		//Load the first position with new data
		gThicknessCtrl.Internal.MediaAnalogValues[0] := gDing.State.xDingLowPieceDetect;

		// If detected in nSensor fast, activate and wait untill slow program to deal with
		IF gDing.State.xMediaToRejectDetected THEN
			gThicknessCtrl.status.Detection.xMediaToRejectDetected := TRUE;
			// Just when the slow program has readed the status.xMediaToReject variable, we can reset the status
		ELSIF gThicknessCtrl.Internal.xMediaToRejectTreated THEN
			gThicknessCtrl.status.Detection.xMediaToRejectDetected := FALSE;
			gThicknessCtrl.Internal.xMediaToRejectTreated := FALSE;
		END_IF

	END_IF

	IF gPhotoCells.status.xInstalled THEN

		ShiftArrayForward(ADR(gThicknessCtrl.Internal.ArrayHeightValues), SIZEOF(gThicknessCtrl.Internal.ArrayHeightValues), SIZEOF(gThicknessCtrl.Internal.ArrayHeightValues[0]), 1, THICK_MAX_UPDATE_VALUES);

		// Photo Cells laser position to heigh detection ctrl
		IF gThicknessCtrl.parameters.xMarginForBendTile THEN
			gThicknessCtrl.Internal.ArrayHeightValues[0] := REAL_TO_UINT(MAX(gPhotoCells.status.rBarsPosition + gThicknessCtrl.Internal.rMarginSafePrintChecked,
														gThicknessCtrl.status.Heigh.rMediaThicknessMargin)*100);

		ELSE
			gThicknessCtrl.Internal.ArrayHeightValues[0] := REAL_TO_UINT(MAX(gPhotoCells.status.rBarsPosition,
														gThicknessCtrl.status.Heigh.rMediaThicknessMargin)*100);
		END_IF

		//Load array of data to avoid loosing information -----------------------------------------
		//Move the array one position
		ShiftArrayForward(ADR(gThicknessCtrl.Internal.MediaArraySensorValues), SIZEOF(gThicknessCtrl.Internal.MediaArraySensorValues), SIZEOF(gThicknessCtrl.Internal.MediaArraySensorValues[0]), 1, THICK_MAX_UPDATE_VALUES);
		//Load the first position with new data
		IF gPhotoCells.status.xTrustPhotocellASignal THEN
			gThicknessCtrl.Internal.MediaArraySensorValues[0] := gPhotoCells.status.xLowPieceDetect;

		ELSE
			gThicknessCtrl.Internal.MediaArraySensorValues[0] := FALSE;
		END_IF

		// If detected in nSensor fast, activate and wait untill slow program to deal with
		IF gPhotoCells.status.xMediaToRejectDetected  THEN
			gThicknessCtrl.status.Detection.xMediaToRejectDetected := TRUE;
			// Just when the slow program has readed the status.xMediaToReject variable, we can reset the status
		ELSIF gThicknessCtrl.Internal.xMediaToRejectTreated THEN
			gThicknessCtrl.status.Detection.xMediaToRejectDetected := FALSE;
			gThicknessCtrl.Internal.xMediaToRejectTreated := FALSE;
		END_IF

	END_IF

	IF gBasicDetectMedia.Status.xInstalled THEN
		// Consider Detection media as an AnalogMedia
		ShiftArrayForward(ADR(gThicknessCtrl.Internal.AnalogHeightValues), SIZEOF(gThicknessCtrl.Internal.AnalogHeightValues), SIZEOF(gThicknessCtrl.Internal.AnalogHeightValues[0]), 1, THICK_MAX_UPDATE_VALUES);
		gThicknessCtrl.Internal.AnalogHeightValues[0] := REAL_TO_UINT(gBasicDetectMedia.Status.rMediaHeigh * 100);

		ShiftArrayForward(ADR(gThicknessCtrl.Internal.MediaDetectionValues), SIZEOF(gThicknessCtrl.Internal.MediaDetectionValues), SIZEOF(gThicknessCtrl.Internal.MediaDetectionValues[0]), 1, THICK_MAX_UPDATE_VALUES);
		//Load the first position with new data
		gThicknessCtrl.Internal.MediaDetectionValues[0] := gBasicDetectMedia.Status.xMediaPresent;
		// TOREVIEW. Need an array per line
		//gThicknessCtrl.Internal.MediaDetectionValuesL1[0] := gBasicDetectMedia.Inputs.xMediaPresentL1;
		//gThicknessCtrl.Internal.MediaDetectionValuesL2[0] := gBasicDetectMedia.Inputs.xMediaPresentL2;
		gThicknessCtrl.Internal.MediaDetectionValuesL1 := gThicknessCtrl.Internal.MediaDetectionValues;

	END_IF

	IF NOT gDing.State.xDingInstalled AND NOT gPhotoCells.status.xInstalled AND NOT gBasicDetectMedia.Status.xInstalled THEN
		//TODO: Here an error should be raised and avoid enter in AutoMode
		gThicknessCtrl.status.Heigh.rMediaHeigh := 0;
	END_IF

	//Load array of data to avoid loosing information -----------------------------------------
	//Move the array one position
	ShiftArrayForward(ADR(xProductDetectValuesL1), SIZEOF(xProductDetectValuesL1), SIZEOF(xProductDetectValuesL1[0]), 1, THICK_MAX_UPDATE_VALUES);
	ShiftArrayForward(ADR(xProductDetectValuesL2), SIZEOF(xProductDetectValuesL2), SIZEOF(xProductDetectValuesL2[0]), 1, THICK_MAX_UPDATE_VALUES);

	// Protection against not assigned pointers
	IF gThicknessCtrl.parameters.Detection.ProductDetect.pMediaInProductDetectL1 = 0 OR
		gThicknessCtrl.parameters.Detection.ProductDetect.pMediaInProductDetectL2 = 0 THEN
		RETURN;
	END_IF

	//Load the first position with new data
	xMediaInProductDetectL1 ACCESS gThicknessCtrl.parameters.Detection.ProductDetect.pMediaInProductDetectL1;
	xMediaInProductDetectL2 ACCESS gThicknessCtrl.parameters.Detection.ProductDetect.pMediaInProductDetectL2;

	iReasonForMediaInProductDetect.0 := xMediaInProductDetectL1;
	iReasonForMediaInProductDetect.1 := xMediaInProductDetectL2;
	gThicknessCtrl.status.Detection.xMediaInProductDetect := iReasonForMediaInProductDetect > 0;

	xProductDetectValuesL1[0] := xMediaInProductDetectL1;
	xProductDetectValuesL2[0] := xMediaInProductDetectL2;

	gThicknessCtrl.Internal.ProductDetectValuesL1 := xProductDetectValuesL1;
	gThicknessCtrl.Internal.ProductDetectValuesL2 := xProductDetectValuesL2;

	//////////////////
	xMountedMedia := gPhotoCells.Alarms.xMountedTile OR gDing.Alarms.xMountedTile;
	IF EDGEPOS(xMountedMedia) THEN
		gThicknessCtrl.status.Belt.rBeltPositionMmInit := gAxis[gBelt.parameters.IndexAxis].Status.ActPosition;
		gThicknessCtrl.status.Belt.rBeltSpeed := gAxis[gBelt.parameters.IndexAxis].Status.ActVelocity;
	END_IF

	IF xMountedMedia AND EDGENEG(gAxis[gBelt.parameters.IndexAxis].Status.PLCopenState.ContinuousMotion) THEN
		gThicknessCtrl.status.Belt.rBeltPositionMmFinal := gAxis[gBelt.parameters.IndexAxis].Status.ActPosition;
	END_IF

END_PROGRAM
```

#### ThickCtrl_Fast.var
```iecst
VAR
	RTInfo_0 : RTInfo;
	rPeriode : REAL := 0; (*Cycle time in microseconds. Read just in INIT. NEVER Write over it!!!*)
	iReasonForMediaInProductDetect : USINT;
	xProductDetectValuesL1 : ARRAY[0..THICK_MAX_UPDATE_VALUES] OF BOOL;
	xProductDetectValuesL2 : ARRAY[0..THICK_MAX_UPDATE_VALUES] OF BOOL;
	xMediaInProductDetectL1 : REFERENCE TO BOOL;
	xMediaInProductDetectL2 : REFERENCE TO BOOL;
END_VAR
VAR RETAIN
	BeltDriveUnit : DriveUnitMngr;
END_VAR
VAR
	xMountedMedia : BOOL; (*Previously as an input, now ThicknessCtrl reads the value from AnalogCtrl and ArrayCtrl*)
END_VAR
```

### Program Logical/ExtPack/_Media/ThicknessCtrl/ThicknessCtrl_v2/ThickReadEnergy (IEC)

#### ThickReadEnergy.st - Implementation code
```iecst
(********************************************************************
 * COPYRIGHT -- EFI
 ********************************************************************
 * Program: ThickReadEnergy from Original BR& LibFileIO1_ST
 * File: ThickReadEnergy.st
 * Author: EFI
 * Created: February 24, 2023
 ********************************************************************
 * Implementation of program Handling
 ********************************************************************)

PROGRAM _INIT

	(* device name for different function blocks needed (choose yourself) *)
	strcpy( ADR(Handling.Data.Device), ADR('LOCAL_DEV') );
	(* perameter string, layout see in the online help by function block "devlink" *)
	strcpy( ADR(Handling.Data.Parameter), ADR('"/DEVICE=C:/EnergyData') );

	(* predefine filenames *)
	strcpy( ADR(Handling.Data.FileName), ADR('TestHex.bin'));

END_PROGRAM

(******************************************)
(* cyclic program                         *)
(******************************************)
PROGRAM _CYCLIC

	// Conexion with gThicknessCtrl
	IF EDGEPOS(gThicknessCtrl.parSw.Dry.xReadFile) THEN
		Handling.Command.bReadExFile := TRUE;
	ELSIF EDGENEG(Handling.Command.bReadExFile) THEN
		gThicknessCtrl.parSw.Dry.xReadFile := FALSE;
	END_IF
	gThicknessCtrl.status.iReadEnergyFileStep := Handling.Data.Step;

	CASE Handling.Data.Step OF

		0:  (* link (create) a file device *)
			Handling.Functionblock.DevLink_0.enable := 1;
			Handling.Functionblock.DevLink_0.pDevice := ADR(Handling.Data.Device);  (* name of the device, which is needed for other functionblocks *)
			Handling.Functionblock.DevLink_0.pParam := ADR(Handling.Data.Parameter);  (* devicepath *)
			Handling.Functionblock.DevLink_0;  (* call the function*)

			IF Handling.Functionblock.DevLink_0.status = 0 THEN  (* DevLink successful *)
				Handling.Data.Step := 1;  (* next Step*)
			ELSIF Handling.Functionblock.DevLink_0.status = ERR_FUB_BUSY THEN  (* DevLink not finished -> redo *)
				(* Busy *)
			ELSIF Handling.Functionblock.DevLink_0.status = fiERR_SYSTEM THEN  (* DevLink error = fiERR_SYSTEM -> detailed info with function "FileIoGetSysError" *)
				(* get detail errorinformation *)
				Error := FileIoGetSysError();
				(* Goto Error Step *)
				Handling.Data.Step := 255;
			ELSE  (* Goto Error Step *)
				Handling.Data.Step := 255;
			END_IF

		1:  (* Wait and comannd step *)
			IF Handling.Command.bReadExFile = 1 THEN
				(* read data to variable "Handling.Data.ReadData"
				   from the file with the name of the variable "Handling.Data.FileName" *)
				Handling.Data.Step := 40;  (* next Step*)

			END_IF

		(***********************************************************************************************)
		40:	(* open file for read access *)
			Handling.Functionblock.FileOpen_0.enable := 1;
			Handling.Functionblock.FileOpen_0.pDevice := ADR(Handling.Data.Device);  (* name of the linked device *)
			Handling.Functionblock.FileOpen_0.pFile :=  ADR(Handling.Data.FileName);  (* name of the file *)
			Handling.Functionblock.FileOpen_0.mode := fiREAD_ONLY;  (* read access *)
			Handling.Functionblock.FileOpen_0;  (* call the function*)

			IF Handling.Functionblock.FileOpen_0.status = 0 THEN  (* FileOpen successful *)
				Handling.Data.Step := 41;  (* next Step*)
			ELSIF Handling.Functionblock.FileOpen_0.status = ERR_FUB_BUSY THEN  (* FileOpen not finished -> redo *)
				(* Busy *)
			ELSE  (* Goto Error Step *)
				Handling.Data.Step := 255;
			END_IF

		41: (* read data from file *)
			Handling.Functionblock.FileReadEx_0.enable := 1;
			Handling.Functionblock.FileReadEx_0.ident := Handling.Functionblock.FileOpen_0.ident;  (* ident of the previous "FileOpen" *)
			Handling.Functionblock.FileReadEx_0.offset := 0;  (* start at the beginning of the file *)
			Handling.Functionblock.FileReadEx_0.pDest := ADR(Handling.Data.ReadDataHex);  (* adress of the destination of reaaded datas *)
			Handling.Functionblock.FileReadEx_0.len := SIZEOF( Handling.Data.ReadDataHex);  (* lenght of data, which should be readed *)
			Handling.Functionblock.FileReadEx_0;  (* call the function*)

			IF Handling.Functionblock.FileReadEx_0.status = 0 THEN  (* FileReadEx successful *)
				(* Handling.Functionblock.FileReadEx_0.bytesread includes the lenght of the readed data *)
				Handling.Data.Step := 42;  (* next Step*)
			ELSIF Handling.Functionblock.FileReadEx_0.status = ERR_FUB_BUSY THEN  (* FileReadEx not finished -> redo *)
				(* Busy *)
			ELSE  (* Goto Error Step *)
				Handling.Data.Step := 255;
			END_IF

		42:	 (* close file, because of limited number of available file handles on the system *)
			Handling.Functionblock.FileClose_0.enable := 1;
			Handling.Functionblock.FileClose_0.ident := Handling.Functionblock.FileOpen_0.ident; (* ident for FileCreate-functionblock*)
			Handling.Functionblock.FileClose_0;  (* call the function*)

			IF Handling.Functionblock.FileClose_0.status = 0 THEN  (* FileClose successful *)
				Handling.Data.Step := 1;  (* next Step*)
				Handling.Command.bReadExFile := 0;  (* clear command *)

				// Assgination to gThicknessCtrl
				gThicknessCtrl.parameters.ContinuousMedia.Energy.iPower := Handling.Data.ReadDataHex;

				Handling.Command.bReadExFile := FALSE;  (* clear command *)

			ELSIF Handling.Functionblock.FileClose_0.status = ERR_FUB_BUSY THEN  (* FileClose not finished -> redo *)
				(* Busy *)
			ELSE  (* Goto Error Step *)
				Handling.Data.Step := 255;
			END_IF

		(***********************************************************************************************)
		255:  (* Here some error Handling has to be implemented *)

	END_CASE

END_PROGRAM
```

#### ThickReadEnergy.typ - Local data types
```iecst
(********************************************************************
 * COPYRIGHT -- Bernecker + Rainer
 ********************************************************************
 * Program: FileHandling
 * File: FileHandling.typ
 * Author: Bernecker + Rainer
 * Created: April 16, 2009
 ********************************************************************
 * Local data types of program FileHandling
 ********************************************************************)

TYPE
	FileHandling_Functionblock_typ : 	STRUCT
		DevLink_0 : DevLink; (*Functionblock DevLink()*)
		FileClose_0 : FileClose; (*Functionblock FileClose()*)
		FileOpen_0 : FileOpen; (*Functionblock FileOpen()*)
		FileReadEx_0 : FileReadEx; (*Functionblock FileReadEx()*)
	END_STRUCT;
	FileHandling_Data_typ : 	STRUCT
		FileName : STRING[32]; (*filename for command bCreateFile, bDeleteFile, bWriteFile, bReadFile, bReadExFile, bCopyFile, bRenameFile*)
		Device : STRING[32]; (*device name*)
		Parameter : STRING[80]; (*parameterstring for FUB DevLink()*)
		ReadDataHex : ARRAY[0..THICKENERGY_MAX_PROCESS_ITEMS,0..THICKENERGY_MAX_CROSS_ITEMS]OF USINT; (*readed data from command bReadFile and bReadExFile*)
		Step : USINT; (*step variable (255 = error step)*)
	END_STRUCT;
	FileHandling_Command_typ : 	STRUCT
		bReadExFile : BOOL; (*Command: read data from file*)
	END_STRUCT;
	FileHandling_typ : 	STRUCT
		Command : FileHandling_Command_typ; (*Command structure*)
		Data : FileHandling_Data_typ; (*Data structure*)
		Functionblock : FileHandling_Functionblock_typ; (*FUB structure*)
	END_STRUCT;
END_TYPE
```

### Program Logical/ExtPack/_Media/ThicknessCtrl/ThicknessCtrlSim/ThicknessCtrlSim_v1/ThicknessCtrlSim (IEC)

#### ThicknessCtrlSim.var - Local variables
```iecst
VAR
	xMediaTracking : REFERENCE TO ARRAY[0..iMAXTRACKINGARRAY] OF USINT; (*Matrix with the information about if there is Media in the position. Each position corresponds to a cm. Bit 0: L1 , Bit 1 L2*)
	iDistanceWorkEmptyBelt : REFERENCE TO UINT;
	iIndexMediaTrack : UINT;
END_VAR
```

### Program Logical/ExtPack/_Tools/SimUseRegister/SimUseRegister_1/SimUseRegister (IEC) - Cyclic code

#### SimUseRegister.typ
```iecst
TYPE
	SimRegisterState :
		(
		SIMR_IDLE,
		SIMR_CREATE_MAIN,
		SIMR_CREATING_MAIN,
		SIMR_CREATE_YEAR,
		SIMR_CREATING_YEAR,
		SIMR_CREATE_FILEREG,
		SIMR_CREATING_FILEREG,
		SIMR_IDLE_MAIN,
		SIMR_STOPPED
		);
END_TYPE
```

#### FileHandling.typ - Local data types
```iecst
(********************************************************************
 * COPYRIGHT -- Bernecker + Rainer
 ********************************************************************
 * Program: FileHandling
 * File: FileHandling.typ
 * Author: Bernecker + Rainer
 * Created: April 16, 2009
 ********************************************************************
 * Local data types of program FileHandling
 ********************************************************************)

TYPE
	FileHandling_Functionblock_typ : 	STRUCT
		DevLink_0 : DevLink; (*Functionblock DevLink()*)
		FileCreate_0 : FileCreate; (*Functionblock FileCreate()*)
		FileClose_0 : FileClose; (*Functionblock FileClose()*)
		FileOpen_0 : FileOpen; (*Functionblock FileOpen()*)
		FileWrite_0 : FileWrite; (*Functionblock FileWrite()*)
		FileRead_0 : FileRead; (*Functionblock FileRead()*)
		FileReadEx_0 : FileReadEx; (*Functionblock FileReadEx()*)
		FileCopy_0 : FileCopy; (*Functionblock FileCopy()*)
		FileRename_0 : FileRename; (*Functionblock FileRename()*)
		FileDelete_0 : FileDelete; (*Functionblock FileDelete()*)
	END_STRUCT;
	FileHandling_Data_typ : 	STRUCT
		FileName : STRING[100]; (*filename for command bCreateFile, bDeleteFile, bWriteFile, bReadFile, bReadExFile, bCopyFile, bRenameFile*)
		NewFileName : STRING[100]; (*new filename for command bCopyFile and bRenameFile*)
		Device : STRING[100]; (*device name*)
		Parameter : STRING[100]; (*parameterstring for FUB DevLink()*)
		WriteData : STRING[80]; (*data for command bWriteFile*)
		ReadData : STRING[80]; (*readed data from command bReadFile and bReadExFile*)
		Step : USINT; (*step variable (255 = error step)*)
	END_STRUCT;
	FileHandling_Command_typ : 	STRUCT
		bCreateFile : BOOL; (*Command: create new file*)
		bWriteFile : BOOL; (*Command: write data into file*)
		bReadFile : BOOL; (*Command: read data from file*)
		bReadExFile : BOOL; (*Command: read data from file*)
		bRenameFile : BOOL; (*Command: rename file*)
		bCopyFile : BOOL; (*Command: create a copy of a file*)
		bDeleteFile : BOOL; (*Command: detete a file*)
	END_STRUCT;
	FileHandling_typ : 	STRUCT
		Command : FileHandling_Command_typ; (*Command structure*)
		Data : FileHandling_Data_typ; (*Data structure*)
		Functionblock : FileHandling_Functionblock_typ; (*FUB structure*)
	END_STRUCT;
END_TYPE
```

### Program Logical/ExtPack/_Tools/EventLog/EventLog_v1/EventLogGen (IEC)

#### EventLog.fun
```iecst
FUNCTION GetSeverity : USINT (*Gets severity from EventId (bits 31-30).*)
	VAR_INPUT
		EventID : DINT;
	END_VAR
END_FUNCTION

FUNCTION GetFacility : UINT (*Gets facility from EventId (bits 27-16).*)
	VAR_INPUT
		EventID : DINT;
	END_VAR
END_FUNCTION

FUNCTION GetCode : UINT (*Gets code from EventId (bits 15-0).*)
	VAR_INPUT
		EventID : DINT;
	END_VAR
END_FUNCTION
```

#### EventLog.st
```iecst
(********************************************************************
 * COPYRIGHT -- Bernecker + Rainer
 ********************************************************************
 * PROGRAM: EventLog
 * File: EventLog.st
 * Author: Bernecker + Rainer
 * Created: June, 2015
 ********************************************************************
 * Implementation OF PROGRAM EventLog
 ********************************************************************)

PROGRAM _INIT
	EventLog.Event.EnteredBy := 'UserID';
	brsstrcpy(ADR(EventLog.Event.AdditionalData), ADR('This is an information entry from the user.'));
	EventLog.Event.AdditionalDataSize := brsstrlen(ADR(EventLog.Event.AdditionalData)) + 1;
	EventLog.Event.AdditionalDataFormat := arEVENTLOG_ADDFORMAT_TEXT;
	(*See ArEventLog help for the description of the event id, facilities 0-15 are reserved for customer use.*)
	EventLog.Event.EventID := ArEventLogMakeEventID(Severity := arEVENTLOG_SEVERITY_INFO, Facility := 10, ErrorCode := 1024);
	EventLog.Commands.CreateUserLog := TRUE; //Always try to create after Init. If the logBook exists, error and keep on working

	//Start the Semaphore creation
	SemFifoCreate.enable := TRUE;
	SemFifoCreate.initCount := 0;  (* initial value of the semaphore *)
	SemFifoCreate.maxCount := 1;  (* maximum possible allocation of semaphore *)
	SemFifoCreate();  (* call the function*)

END_PROGRAM

PROGRAM _CYCLIC

	//Wait to create the semaphore
	IF SemIdent = 0 THEN
		IF SemFifoCreate.status = ERR_OK THEN  //SemCreate successful
			SemIdent := SemFifoCreate.ident;  //copy semaphore-ident the a local variable
			SemFifoCreate(enable := FALSE);

			SemRelease( SemIdent );  //release the allocated semaphore
			gEventLogLoader(SemId := SemIdent); //Send the information to the loader
			gEventLogManager(SemId := SemIdent); //Sent the information to the manager
		ELSE
			SemFifoCreate();
			RETURN;
		END_IF
	END_IF

	//Initialize gEventLogLoader
	IF NOT gEventLogLoader.InitDone THEN
		gEventLogLoader();
	END_IF

	//If EventLogManager is not been executed by adding an event, execute it
	gEventLogManager(EventLog := ADR(EventLog));

	CASE EventLog.Data.Step OF
		(*Waits for user input (command).*)
		STEP_WAIT_FOR_INPUT:
			IF EventLog.Commands.CreateUserLog THEN
				EventLog.Commands.CreateUserLog := FALSE;
				EventLog.Data.Step := STEP_GET_LOGBOOK_IDENT;
				EventLog.Data.GetIdentFailNextStep := STEP_CREATE_LOGBOOK;
				EventLog.Data.GetIdentOkNextStep := STEP_WAIT_FOR_INPUT;
				EventLog.Status.execCreateLog:=EventLog.Status.execCreateLog+1;
			ELSIF EventLog.Commands.DeleteUserLog THEN
				EventLog.Commands.DeleteUserLog := FALSE;
				EventLog.Data.Step := STEP_GET_LOGBOOK_IDENT;
				EventLog.Data.GetIdentFailNextStep := STEP_ERROR;
				EventLog.Data.GetIdentOkNextStep := STEP_DELETE_LOGBOOK;
			ELSIF EventLog.Commands.WriteUserEvent THEN
				EventLog.Commands.WriteUserEvent := FALSE;
				EventLog.Data.Step := STEP_GET_LOGBOOK_IDENT;
				EventLog.Data.GetIdentFailNextStep := STEP_ERROR;
				EventLog.Data.GetIdentOkNextStep := STEP_WRITE_EVENT;

				EventLog.Status.execWriteEvent:=EventLog.Status.execWriteEvent+1;
				EventLog.Event.Status := ELOG_STATUS_LOGGING;

			ELSIF EventLog.Commands.ReadLatestEvent THEN
				EventLog.Commands.ReadLatestEvent := FALSE;
				EventLog.Data.Step := STEP_GET_LOGBOOK_IDENT;
				EventLog.Data.GetIdentFailNextStep := STEP_ERROR;
				EventLog.Data.GetIdentOkNextStep := STEP_GET_LATEST_RECORD_ID;
			ELSIF EventLog.Commands.ReadPreviousEvent THEN
				EventLog.Commands.ReadPreviousEvent := FALSE;
				EventLog.Data.Step := STEP_GET_LOGBOOK_IDENT;
				EventLog.Data.GetIdentFailNextStep := STEP_ERROR;
				EventLog.Data.GetIdentOkNextStep := STEP_GET_PREVIOUS_RECORD_ID;
			END_IF

		(*Gets the ident of the user logbook "EFIEvLog".*)
		STEP_GET_LOGBOOK_IDENT:
			IF EventLog.FunctionBlocks.ArEventLogGetIdent_0.Done THEN
				EventLog.FunctionBlocks.ArEventLogGetIdent_0.Execute := FALSE;
				EventLog.Data.Ident := EventLog.FunctionBlocks.ArEventLogGetIdent_0.Ident;
				EventLog.Data.StatusID := ERR_OK;
				EventLog.Data.Step := EventLog.Data.GetIdentOkNextStep;
			ELSIF EventLog.FunctionBlocks.ArEventLogGetIdent_0.Error THEN
				EventLog.FunctionBlocks.ArEventLogGetIdent_0.Execute := FALSE;
				EventLog.Data.StatusID := EventLog.FunctionBlocks.ArEventLogGetIdent_0.StatusID;
				EventLog.Data.Step := EventLog.Data.GetIdentFailNextStep;
			ELSE
				(*Execute the FB only if the ident isn't already set.*)
				IF EventLog.Data.Ident = 0 THEN
					EventLog.FunctionBlocks.ArEventLogGetIdent_0.Name := 'EFIEvLog';
					EventLog.FunctionBlocks.ArEventLogGetIdent_0.Execute := TRUE;
				ELSE
					EventLog.Data.StatusID := ERR_OK;
					EventLog.Data.Step := EventLog.Data.GetIdentOkNextStep;
				END_IF
			END_IF

		(*Creates the user logbook "EFIEvLog".*)
		STEP_CREATE_LOGBOOK:
			IF EventLog.FunctionBlocks.ArEventLogCreate_0.Done THEN
				EventLog.FunctionBlocks.ArEventLogCreate_0.Execute := FALSE;
				EventLog.Data.Ident := EventLog.FunctionBlocks.ArEventLogCreate_0.Ident;
				EventLog.Data.StatusID := ERR_OK;
				EventLog.Data.Step := STEP_WAIT_FOR_INPUT;
			ELSIF EventLog.FunctionBlocks.ArEventLogCreate_0.Error THEN
				EventLog.FunctionBlocks.ArEventLogCreate_0.Execute := FALSE;
				EventLog.Data.StatusID := EventLog.FunctionBlocks.ArEventLogCreate_0.StatusID;
				EventLog.Data.Step := STEP_ERROR;
			ELSE
				EventLog.FunctionBlocks.ArEventLogCreate_0.Name := 'EFIEvLog';
				EventLog.FunctionBlocks.ArEventLogCreate_0.Size := 4096000;
				EventLog.FunctionBlocks.ArEventLogCreate_0.Persistence := arEVENTLOG_PERSISTENCE_PERSIST;
				EventLog.FunctionBlocks.ArEventLogCreate_0.Info := 0;
				EventLog.FunctionBlocks.ArEventLogCreate_0.Execute := TRUE;
			END_IF

		(*Deletes the user logbook "EFIEvLog".*)
		STEP_DELETE_LOGBOOK:
			IF EventLog.FunctionBlocks.ArEventLogDelete_0.Done THEN
				EventLog.FunctionBlocks.ArEventLogDelete_0.Execute := FALSE;
				EventLog.Data.Ident := 0;
				EventLog.Data.StatusID := ERR_OK;
				EventLog.Data.Step := STEP_WAIT_FOR_INPUT;
			ELSIF EventLog.FunctionBlocks.ArEventLogDelete_0.Error THEN
				EventLog.FunctionBlocks.ArEventLogDelete_0.Execute := FALSE;
				EventLog.Data.StatusID := EventLog.FunctionBlocks.ArEventLogDelete_0.StatusID;
				EventLog.Data.Step := STEP_ERROR;
			ELSE
				EventLog.FunctionBlocks.ArEventLogDelete_0.Ident := EventLog.Data.Ident;
				EventLog.FunctionBlocks.ArEventLogDelete_0.Execute := TRUE;
			END_IF

		(*Writes the event set in EventLog.Event to the user logbook "EFIEvLog".*)
		STEP_WRITE_EVENT:
			IF EventLog.FunctionBlocks.ArEventLogWrite_0.Done THEN
				EventLog.FunctionBlocks.ArEventLogWrite_0.Execute := FALSE;
				EventLog.Data.StatusID := ERR_OK;
				EventLog.Data.Step := STEP_WAIT_FOR_INPUT;
				EventLog.Event.Status := ELOG_STATUS_LOGGED;
			ELSIF EventLog.FunctionBlocks.ArEventLogWrite_0.Error THEN
				EventLog.FunctionBlocks.ArEventLogWrite_0.Execute := FALSE;
				EventLog.Data.StatusID := EventLog.FunctionBlocks.ArEventLogWrite_0.StatusID;
				EventLog.Data.Step := STEP_ERROR;
			ELSE
				EventLog.FunctionBlocks.ArEventLogWrite_0.Ident := EventLog.Data.Ident;
				EventLog.Event.EventID := ArEventLogMakeEventID(Severity := EventLog.Event.Severity, Facility := EventLog.Event.Facility, ErrorCode := EventLog.Event.ErrorCode);
				EventLog.FunctionBlocks.ArEventLogWrite_0.EventID := EventLog.Event.EventID;
				EventLog.FunctionBlocks.ArEventLogWrite_0.TimeStamp := 0; (*System timestamp.*)
				EventLog.FunctionBlocks.ArEventLogWrite_0.ObjectID := EventLog.Event.EnteredBy;
				EventLog.FunctionBlocks.ArEventLogWrite_0.OriginRecordID := EventLog.Event.OriginID;
				EventLog.FunctionBlocks.ArEventLogWrite_0.AddDataFormat := EventLog.Event.AdditionalDataFormat;
				EventLog.FunctionBlocks.ArEventLogWrite_0.AddDataSize := EventLog.Event.AdditionalDataSize;
				EventLog.FunctionBlocks.ArEventLogWrite_0.AddData := ADR(EventLog.Event.AdditionalData);
				EventLog.FunctionBlocks.ArEventLogWrite_0.Execute := TRUE;
			END_IF

		(*Gets the id of the latest record in the user logbook "EFIEvLog".*)
		STEP_GET_LATEST_RECORD_ID:
			IF EventLog.FunctionBlocks.ArEventLogGetLatestRecordID_0.Done THEN
				EventLog.FunctionBlocks.ArEventLogGetLatestRecordID_0.Execute := FALSE;
				EventLog.Event.RecordID := EventLog.FunctionBlocks.ArEventLogGetLatestRecordID_0.RecordID;
				EventLog.Data.StatusID := ERR_OK;
				EventLog.Data.Step := STEP_READ_EVENT;
			ELSIF EventLog.FunctionBlocks.ArEventLogGetLatestRecordID_0.Error THEN
				EventLog.FunctionBlocks.ArEventLogGetLatestRecordID_0.Execute := FALSE;
				EventLog.Data.StatusID := EventLog.FunctionBlocks.ArEventLogGetLatestRecordID_0.StatusID;
				EventLog.Data.Step := STEP_ERROR;
			ELSE
				EventLog.FunctionBlocks.ArEventLogGetLatestRecordID_0.Ident := EventLog.Data.Ident;
				EventLog.FunctionBlocks.ArEventLogGetLatestRecordID_0.Execute := TRUE;
			END_IF

		(*Gets the id of the previous record of the given record id (EventLog.Event.RecordID).*)
		STEP_GET_PREVIOUS_RECORD_ID:
			IF EventLog.FunctionBlocks.ArEventLogGetPreviousRecordID_0.Done THEN
				EventLog.FunctionBlocks.ArEventLogGetPreviousRecordID_0.Execute := FALSE;
				EventLog.Event.RecordID := EventLog.FunctionBlocks.ArEventLogGetPreviousRecordID_0.PrevRecordID;
				EventLog.Data.StatusID := ERR_OK;
				EventLog.Data.Step := STEP_READ_EVENT;
			ELSIF EventLog.FunctionBlocks.ArEventLogGetPreviousRecordID_0.Error THEN
				EventLog.FunctionBlocks.ArEventLogGetPreviousRecordID_0.Execute := FALSE;
				EventLog.Data.StatusID := EventLog.FunctionBlocks.ArEventLogGetPreviousRecordID_0.StatusID;
				EventLog.Data.Step := STEP_ERROR;
			ELSE
				EventLog.FunctionBlocks.ArEventLogGetPreviousRecordID_0.Ident := EventLog.Data.Ident;
				EventLog.FunctionBlocks.ArEventLogGetPreviousRecordID_0.RecordID := EventLog.Event.RecordID;
				EventLog.FunctionBlocks.ArEventLogGetPreviousRecordID_0.Execute := TRUE;
			END_IF

		(*Reads the event with the given record id from the to user logbook "EFIEvLog".*)
		STEP_READ_EVENT:
			IF EventLog.FunctionBlocks.ArEventLogRead_0.Done THEN
				EventLog.FunctionBlocks.ArEventLogRead_0.Execute := FALSE;
				EventLog.Event.AdditionalDataFormat := EventLog.FunctionBlocks.ArEventLogRead_0.AddDataFormat;
				EventLog.Event.AdditionalDataSize := EventLog.FunctionBlocks.ArEventLogRead_0.AddDataSize;
				EventLog.Event.TimeStamp := EventLog.FunctionBlocks.ArEventLogRead_0.TimeStamp;
				EventLog.Event.OriginID := EventLog.FunctionBlocks.ArEventLogRead_0.OriginRecordID;
				EventLog.Data.StatusID := ERR_OK;
				EventLog.Event.ErrorNumber := 0;
				EventLog.Event.Customer := ArEventLogIsCustomerArea(EventID := EventLog.FunctionBlocks.ArEventLogRead_0.EventID);
				EventLog.Event.Severity := GetSeverity(EventID := EventLog.FunctionBlocks.ArEventLogRead_0.EventID);
				EventLog.Event.Code := GetCode(EventID := EventLog.FunctionBlocks.ArEventLogRead_0.EventID);
				EventLog.Event.Facility := GetFacility(EventID := EventLog.FunctionBlocks.ArEventLogRead_0.EventID);
				IF EventLog.FunctionBlocks.ArEventLogRead_0.StatusID = arEVENTLOG_WRN_NO_EVENTID THEN
					(*The given record id is not an event id record. Invoke ArEventLogReadErrorNumber to read the error number and the severity.*)
					EventLog.Data.Step := STEP_READ_ERROR_NUMBER;
				ELSIF EventLog.Event.AdditionalDataSize > 0 THEN
					EventLog.Data.Step := STEP_READ_ADDITIONAL_DATA;
				ELSE
					EventLog.Data.Step := STEP_READ_OBJECT_ID;
				END_IF
			ELSIF EventLog.FunctionBlocks.ArEventLogRead_0.Error THEN
				EventLog.FunctionBlocks.ArEventLogRead_0.Execute := FALSE;
				EventLog.Data.StatusID := EventLog.FunctionBlocks.ArEventLogRead_0.StatusID;
				EventLog.Data.Step := STEP_ERROR;
			ELSE
				EventLog.FunctionBlocks.ArEventLogRead_0.Ident := EventLog.Data.Ident;
				EventLog.FunctionBlocks.ArEventLogRead_0.RecordID := EventLog.Event.RecordID;
				EventLog.FunctionBlocks.ArEventLogRead_0.Execute := TRUE;
			END_IF

		(*Reads the error number event with the given record id from the user logbook "EFIEvLog".*)
		STEP_READ_ERROR_NUMBER:
			IF EventLog.FunctionBlocks.ArEventLogReadErrorNumber_0.Done THEN
				EventLog.FunctionBlocks.ArEventLogReadErrorNumber_0.Execute := FALSE;
				EventLog.Event.ErrorNumber := EventLog.FunctionBlocks.ArEventLogReadErrorNumber_0.ErrorNumber;
				EventLog.Event.Severity := EventLog.FunctionBlocks.ArEventLogReadErrorNumber_0.Severity;
				EventLog.Data.StatusID := ERR_OK;
				IF EventLog.Event.AdditionalDataSize > 0 THEN
					EventLog.Data.Step := STEP_READ_ADDITIONAL_DATA;
				ELSE
					EventLog.Data.Step := STEP_READ_OBJECT_ID;
				END_IF
			ELSIF EventLog.FunctionBlocks.ArEventLogReadErrorNumber_0.Error THEN
				EventLog.FunctionBlocks.ArEventLogReadErrorNumber_0.Execute := FALSE;
				EventLog.Data.StatusID := EventLog.FunctionBlocks.ArEventLogReadErrorNumber_0.StatusID;
				EventLog.Data.Step := STEP_ERROR;
			ELSE
				EventLog.FunctionBlocks.ArEventLogReadErrorNumber_0.Ident := EventLog.Data.Ident;
				EventLog.FunctionBlocks.ArEventLogReadErrorNumber_0.RecordID := EventLog.Event.RecordID;
				EventLog.FunctionBlocks.ArEventLogReadErrorNumber_0.Execute := TRUE;
			END_IF

		(*Reads the additional data of the event with the given record id from the user logbook "EFIEvLog".*)
		STEP_READ_ADDITIONAL_DATA:
			IF EventLog.FunctionBlocks.ArEventLogReadAddData_0.Done THEN
				EventLog.FunctionBlocks.ArEventLogReadAddData_0.Execute := FALSE;
				EventLog.Event.AdditionalDataSize := EventLog.FunctionBlocks.ArEventLogReadAddData_0.AddDataSize;
				EventLog.Data.StatusID := ERR_OK;
				EventLog.Data.Step := STEP_READ_OBJECT_ID;
			ELSIF EventLog.FunctionBlocks.ArEventLogReadAddData_0.Error THEN
				EventLog.FunctionBlocks.ArEventLogReadAddData_0.Execute := FALSE;
				EventLog.Data.StatusID := EventLog.FunctionBlocks.ArEventLogReadAddData_0.StatusID;
				EventLog.Data.Step := STEP_ERROR;
			ELSE
				EventLog.FunctionBlocks.ArEventLogReadAddData_0.Ident := EventLog.Data.Ident;
				EventLog.FunctionBlocks.ArEventLogReadAddData_0.RecordID := EventLog.Event.RecordID;
				EventLog.FunctionBlocks.ArEventLogReadAddData_0.BytesToRead := SIZEOF(EventLog.Event.AdditionalData);
				EventLog.FunctionBlocks.ArEventLogReadAddData_0.AddData := ADR(EventLog.Event.AdditionalData);
				EventLog.FunctionBlocks.ArEventLogReadAddData_0.Execute := TRUE;
			END_IF

		(*Reads the object id of the event with the given record id from the user logbook "EFIEvLog".*)
		STEP_READ_OBJECT_ID:
			IF EventLog.FunctionBlocks.ArEventLogReadObjectID_0.Done THEN
				EventLog.FunctionBlocks.ArEventLogReadObjectID_0.Execute := FALSE;
				EventLog.Event.EnteredBy := EventLog.FunctionBlocks.ArEventLogReadObjectID_0.ObjectID;
				EventLog.Data.StatusID := ERR_OK;
				EventLog.Data.Step := STEP_WAIT_FOR_INPUT;
			ELSIF EventLog.FunctionBlocks.ArEventLogReadObjectID_0.Error THEN
				EventLog.FunctionBlocks.ArEventLogReadObjectID_0.Execute := FALSE;
				EventLog.Data.StatusID := EventLog.FunctionBlocks.ArEventLogReadObjectID_0.StatusID;
				EventLog.Data.Step := STEP_ERROR;
			ELSE
				EventLog.FunctionBlocks.ArEventLogReadObjectID_0.Ident := EventLog.Data.Ident;
				EventLog.FunctionBlocks.ArEventLogReadObjectID_0.RecordID := EventLog.Event.RecordID;
				EventLog.FunctionBlocks.ArEventLogReadObjectID_0.Execute := TRUE;
			END_IF

		STEP_ERROR:
		(*Do some error handling here.*)
	END_CASE

	EventLog.FunctionBlocks.ArEventLogCreate_0;
	EventLog.FunctionBlocks.ArEventLogDelete_0;
	EventLog.FunctionBlocks.ArEventLogWrite_0;
	EventLog.FunctionBlocks.ArEventLogGetIdent_0;
	EventLog.FunctionBlocks.ArEventLogGetLatestRecordID_0;
	EventLog.FunctionBlocks.ArEventLogGetPreviousRecordID_0;
	EventLog.FunctionBlocks.ArEventLogReadAddData_0;
	EventLog.FunctionBlocks.ArEventLogReadErrorNumber_0;
	EventLog.FunctionBlocks.ArEventLogReadObjectID_0;
	EventLog.FunctionBlocks.ArEventLogRead_0;
END_PROGRAM

(*See ArEventLog help for the description of the event id format!*)

(*Gets severity from EventId (bits 31-30).*)
FUNCTION GetSeverity
	IF ArEventLogIsError(EventID := EventID) THEN
		GetSeverity := arEVENTLOG_SEVERITY_ERROR;
	ELSIF ArEventLogIsWarning(EventID := EventID) THEN
		GetSeverity := arEVENTLOG_SEVERITY_WARNING;
	ELSIF ArEventLogIsInformation(EventID := EventID) THEN
		GetSeverity := arEVENTLOG_SEVERITY_INFO;
	ELSIF ArEventLogIsSuccess(EventID := EventID) THEN
		GetSeverity := arEVENTLOG_SEVERITY_SUCCESS;
	END_IF
END_FUNCTION

(*Gets code from EventId (bits 15-0).*)
FUNCTION GetCode
	GetCode := DINT_TO_UINT(EventID);
END_FUNCTION

(*Gets facility from EventId (bits 27-16).*)
FUNCTION GetFacility
	GetFacility := DINT_TO_UINT(SHR(EventID, 16) AND 16#0FFF);
END_FUNCTION
```

### Library Logical/ExtPack/_Tools/EventLog/EventLog_v1/EvLogLib (IEC)

#### EvLog.typ
```iecst
TYPE
	EventLogSeverity_enum :
		(
		ELOG_SEVERITY_INFO,
		ELOG_SEVERITY_WARNING,
		ELOG_SEVERITY_ERROR,
		ELOG_SEVERITY_SUCCESS
		);
	EventLogStatus_enum :
		(
		ELOG_STATUS_CREATED,
		ELOG_STATUS_QUEUED,
		ELOG_STATUS_LOGGING,
		ELOG_STATUS_LOGGED
		);
	EventLogCreatedBy_enum :
		(
		ELOG_TYPE_GENERAL,
		ELOG_TYPE_BAR,
		ELOG_TYPE_BLOCK,
		ELOG_TYPE_SIMPLEBLOCK,
		ELOG_TYPE_BELT,
		ELOG_TYPE_LED,
		ELOG_TYPE_TRANS_VACUUM,
		ELOG_TYPE_NONCRASH,
		ELOG_TYPE_NIR,
		ELOG_TYPE_ARCLAMP,
		ELOG_TYPE_DETECTION,
		ELOG_TYPE_EHD,
		ELOG_TYPE_PAIRED_ICLA
		);
	EventLogStatus_typ : 	STRUCT
		Location : USINT;
		Source : BOOL;
		xQueued : BOOL;
	END_STRUCT;
	EventLog_typ : 	STRUCT
		Severity : EventLogSeverity_enum := ELOG_SEVERITY_INFO; (*Severity of the last event (read).*)
		Facility : UINT; (*Facility of the last event (read).*)
		ErrorCode : UINT; (*Error number of the event- set when the read event is no event id event (read).*)
		Source : EventLogCreatedBy_enum := ELOG_TYPE_GENERAL;
		Status : EventLogStatus_enum := ELOG_STATUS_CREATED;
		Text : STRING[129];
		pMyDir : UDINT;
	END_STRUCT;
	EventLogFifoFB : 	STRUCT
		fDelete : fifoDelete;
		fWrite : fifoWrite;
		fRead : fifoRead;
		fGetInfo : fifoGetInfo;
		fCreate : fifoCreate;
	END_STRUCT;
	GenEventLog_typ : 	STRUCT  (*Event handling.*)
		Commands : EventLog_Commands_typ; (*Event handling user commands.*)
		Data : EventLog_Data_typ; (*Event handling data for state machine.*)
		Status : EventLog_Status_typ; (*Event handling event description.*)
		Event : EventLog_Event_typ; (*Event handling event description.*)
		FunctionBlocks : EventLog_FunctionBlocks_typ; (*Event handling used functionblocks.*)
	END_STRUCT;
	EventLog_Commands_typ : 	STRUCT
		CreateUserLog : BOOL; (*Creates the user logbook "EFIEvLog" in USERROM.*)
		DeleteUserLog : BOOL; (*Deletes the user logbook "EFIEvLog".*)
		WriteUserEvent : BOOL; (*Writes a user event into the user logbook "EFIEvLog". *)
		ReadLatestEvent : BOOL; (*Reads the latest event of the user logbook "EFIEvLog".*)
		ReadPreviousEvent : BOOL; (*Reads the previous event (of the given record id) of the user logbook "UserEvLog".*)
	END_STRUCT;
	EventLog_Status_typ : 	STRUCT
		execWriteEvent : UDINT; (*Status information for STEP_ERROR.*)
		execCreateLog : UDINT; (*Status information for STEP_ERROR.*)
	END_STRUCT;
	EventLog_Data_typ : 	STRUCT
		Step : EventLogSteps; (*Current step. STEP_ERROR must be manually reset (STEP_WAIT_FOR_INPUT).*)
		Ident : ArEventLogIdentType; (*Ident of the logbook "EFIEvLog".*)
		StatusID : DINT; (*Status information for STEP_ERROR.*)
		GetIdentOkNextStep : EventLogSteps; (*Internal helper for state machine.*)
		GetIdentFailNextStep : EventLogSteps; (*Internal helper for state machine.*)
	END_STRUCT;
	EventLog_Event_typ : 	STRUCT
		Severity : USINT; (*Severity of the last event (read).*)
		Customer : BOOL; (*Customer bit of the last event (read).*)
		Facility : UINT; (*Facility of the last event (read).*)
		Code : UINT; (*Code of the last event (read).*)
		EventID : DINT; (*EventID for write event (write - is not set by reading an event).*)
		ErrorCode : UINT; (*Error number of the event- set when the read event is no event id event (read).*)
		ErrorNumber : UDINT; (*Error number of the event- set when the read event is no event id event (read).*)
		EnteredBy : STRING[36]; (*User/object identification (read/write - optional).*)
		OriginID : ArEventLogRecordIDType; (*Record id of the origin record (read/write - optional).*)
		RecordID : ArEventLogRecordIDType; (*Record id of the event to read (read - set automatically).*)
		TimeStamp : ArEventLogTimeStampType;
		Status : EventLogStatus_enum;
		AdditionalDataSize : UDINT; (*Size of the additional data (read/write - optional)*)
		AdditionalDataFormat : USINT; (*Format of the additional data (read/write)*)
		AdditionalData : ARRAY[0..128]OF USINT; (*Additional data (read/write)*)
	END_STRUCT;
	EventLog_FunctionBlocks_typ : 	STRUCT
		ArEventLogCreate_0 : ArEventLogCreate;
		ArEventLogDelete_0 : ArEventLogDelete;
		ArEventLogGetIdent_0 : ArEventLogGetIdent;
		ArEventLogGetLatestRecordID_0 : ArEventLogGetLatestRecordID;
		ArEventLogGetPreviousRecordID_0 : ArEventLogGetPreviousRecordID;
		ArEventLogWrite_0 : ArEventLogWrite;
		ArEventLogRead_0 : ArEventLogRead;
		ArEventLogReadErrorNumber_0 : ArEventLogReadErrorNumber;
		ArEventLogReadAddData_0 : ArEventLogReadAddData;
		ArEventLogReadObjectID_0 : ArEventLogReadObjectID;
	END_STRUCT;
	EventLogSteps :
		(
		STEP_WAIT_FOR_INPUT := 0,
		STEP_CREATE_LOGBOOK := 1,
		STEP_DELETE_LOGBOOK := 2,
		STEP_GET_LOGBOOK_IDENT := 3,
		STEP_WRITE_EVENT := 4,
		STEP_READ_EVENT := 5,
		STEP_READ_ERROR_NUMBER := 6,
		STEP_READ_ADDITIONAL_DATA := 7,
		STEP_READ_OBJECT_ID := 8,
		STEP_GET_LATEST_RECORD_ID := 9,
		STEP_GET_PREVIOUS_RECORD_ID := 10,
		STEP_ERROR := 255
		);
END_TYPE
```

#### EvLogLib.fun
```iecst
FUNCTION GetSeverity : USINT
	VAR_INPUT
		Severity : EventLogSeverity_enum;
	END_VAR
END_FUNCTION

FUNCTION GetGroupName : BOOL
	VAR_INPUT
		GenEventLog : REFERENCE TO GenEventLog_typ;
		EventLog : REFERENCE TO EventLog_typ;
	END_VAR
END_FUNCTION

{REDUND_ERROR} FUNCTION_BLOCK EventLoader (*TODO: Add your comment here*) (*$GROUP=User,$CAT=User,$GROUPICON=User.png,$CATICON=User.png*)
	VAR_INPUT
		EventData : REFERENCE TO EventLog_typ;
		SemId : UDINT; (*Semaphore identifier*)
	END_VAR
	VAR_OUTPUT
		InitDone : BOOL := FALSE; (*0*)
	END_VAR
	VAR
		execAdd : UDINT; (*0*)
		statusGetIdent : UDINT := 0; (*0*)
		ident : UDINT := 0; (*0*)
		pEventData : UDINT;
		Fifo : EventLogFifoFB; (*0*)
		InternalEventData : {REDUND_UNREPLICABLE} EventLog_typ;
		uiSemStatus : UINT;
	END_VAR
END_FUNCTION_BLOCK

{REDUND_ERROR} FUNCTION_BLOCK EventManager (*TODO: Add your comment here*) (*$GROUP=User,$CAT=User,$GROUPICON=User.png,$CATICON=User.png*)
	VAR_INPUT
		EventLog : REFERENCE TO GenEventLog_typ;
		SemId : UDINT; (*Semaphore identifier*)
	END_VAR
	VAR
		workEventData : REFERENCE TO EventLog_typ; (*The eventData to work with the program to write*)
		execReview : UDINT; (*0*)
		execEventData : UDINT; (*0*)
		execLogging : UDINT; (*0*)
		statusGetIdent : UDINT := 0; (*0*)
		ident : UDINT := 0; (*0*)
		xLoggingEvent : BOOL := FALSE; (*0*)
		Init : BOOL := FALSE; (*0*)
		Fifo : EventLogFifoFB; (*0*)
		pEventData : UDINT;
		EventDataRead : REFERENCE TO EventLog_typ;
		InternalEventData : {REDUND_UNREPLICABLE} EventLog_typ;
		uiSemStatus : UINT;
	END_VAR
END_FUNCTION_BLOCK
```

#### EventLoader.st
```iecst
(* TODO: Add your comment here *)
FUNCTION_BLOCK EventLoader

	//If not Semaphore, return
	IF SemId = 0 THEN
		RETURN;
	END_IF

	//Create the FIFO at init. Return while creating the FIFO
	IF NOT InitDone THEN
		Fifo.fCreate();
		IF Fifo.fCreate.status = ERR_OK THEN
			Fifo.fCreate.enable := FALSE;
			ident:=Fifo.fCreate.ident;
			InitDone:=TRUE;
		ELSIF Fifo.fCreate.status = fifoERR_FIFO_ALREADY_EXISTS THEN
			statusGetIdent:=fifoGetIdent(pFifo:= ADR('EvLog'), pIdent:=ADR(ident));
			InitDone:=TRUE;
		ELSIF Fifo.fCreate.status <> ERR_FUB_BUSY THEN
			Fifo.fCreate.enable := TRUE;
			Fifo.fCreate.pFifo := ADR('EvLog'); //Name of the FIFO
			Fifo.fCreate.size := 60 * SIZEOF(EventLog_typ); // XX elements size
			Fifo.fCreate.mode := fifoMODE_WRITE_UNTIL_FULL;
		END_IF
		RETURN;
	END_IF

	//If nothing to Load, return
	IF ADR(EventData) = 0 THEN
		RETURN;
	END_IF

	//Try to Acquire the Semaphore
	uiSemStatus := SemAcquire(SemId);
	IF uiSemStatus = semERR_NOT_FREE THEN
		RETURN;
	END_IF

	Fifo.fGetInfo.enable:=TRUE;
	Fifo.fGetInfo.ident := ident;
	Fifo.fGetInfo();

	EventData.Status := ELOG_STATUS_QUEUED;
	EventData.pMyDir := ADR(EventData);

	//Add an Event to the Stack
	Fifo.fWrite.enable:=TRUE;
	Fifo.fWrite.pData := ADR(EventData);
	Fifo.fWrite.ident := ident;
	Fifo.fWrite.size := SIZEOF(EventLog_typ);
	Fifo.fWrite();

	pEventData:=ADR(EventData);

	IF Fifo.fWrite.status = ERR_OK THEN
		Fifo.fWrite.enable:=FALSE;
		//EventData.Status := ELOG_STATUS_QUEUED;
	END_IF

	InternalEventData:=EventData;

	//Release the Semaphore
	SemRelease(SemId);

	execAdd := execAdd +1;

END_FUNCTION_BLOCK
```

### TraySimGen.var
```iecst
VAR
	iTraySimIndex : USINT;
END_VAR
```

### Program Logical/ExtPack/_Tools/TestBench/TraySim/TraySim_v1/InitTraySim (IEC)

#### Cyclic.st - Cyclic code
```iecst
PROGRAM _CYCLIC
	(* Insert code here *)
	iTraySimIndex := 1;

END_PROGRAM
```

### Program Logical/ExtPack/_Tools/TestBench/TraySim/TraySim_v1/TraySim

#### Main.st
```iecst
PROGRAM _CYCLIC
	(* Insert code here *)

	trayData  ACCESS ADR(gTraySim[iTraySimIndex]);

	//Remove both orders if two different orders at the same time
	IF trayData.Commands.ToIn AND trayData.Commands.ToOut THEN
		trayData.Commands.ToIn := FALSE;
		trayData.Commands.ToOut := FALSE;
	END_IF

	IF EDGEPOS(trayData.Commands.ToIn) THEN xReboundedIn := FALSE; END_IF
	ton_ToIn.IN:= trayData.Commands.ToIn AND NOT xReboundedIn;
	ton_ToIn.PT := t#1s;
	ton_ToIn();

	ton_ReboundIn.IN := trayData.State.InPosition AND trayData.Commands.ReboundToIn;
	ton_ReboundIn.PT := t#500ms;
	ton_ReboundIn();

	IF EDGEPOS(trayData.Commands.ToOut) THEN xReboundedOut := FALSE; END_IF
	ton_ToOut.IN:= trayData.Commands.ToOut AND NOT xReboundedOut;
	ton_ToOut.PT := t#1s;
	ton_ToOut();

	ton_ReboundOut.IN := trayData.State.OutPosition AND trayData.Commands.ReboundToOut;
	ton_ReboundOut.PT := t#500ms;
	ton_ReboundOut();

	//In sensor
	IF NOT trayData.Commands.UnplugInSensor THEN
		IF ton_ToIn.Q THEN
			trayData.State.InPosition := TRUE;
		ELSIF trayData.Commands.ToOut THEN
			trayData.State.InPosition := FALSE;
		ELSIF ton_ReboundIn.Q THEN
			xReboundedIn := TRUE;
			trayData.State.InPosition := FALSE;
		END_IF
	ELSE
		trayData.State.InPosition := FALSE;
	END_IF

	IF trayData.Commands.ResetIn THEN
		trayData.Commands.ResetIn := FALSE;
		trayData.State.InPosition := FALSE;
	END_IF

	//Out sensor
	IF NOT trayData.Commands.UnplugOutSensor THEN
		IF ton_ToOut.Q THEN
			trayData.State.OutPosition := TRUE;
		ELSIF trayData.Commands.ToIn THEN
			trayData.State.OutPosition := FALSE;
		ELSIF ton_ReboundOut.Q THEN
			xReboundedOut := TRUE;
			trayData.State.OutPosition := FALSE;
		END_IF
	ELSE
		trayData.State.OutPosition := FALSE;
	END_IF

	IF trayData.Commands.ResetOut THEN
		trayData.Commands.ResetOut := FALSE;
		trayData.State.OutPosition := FALSE;
	END_IF

	iTraySimIndex := iTraySimIndex + 1;

END_PROGRAM
```

### Package Logical/ExtPack/_Comms/ModbusComms - Modbus Ctrl Logic package

### Package Logical/ExtPack/_Comms/ModbusComms/ModbusComms_v1 - Modbus Ctrl Logic package

### Program Logical/ExtPack/_Comms/ModbusComms/ModbusComms_v1/ServModbus (IEC) - Slave modbus cyclic task

#### Slave_mbus.st - Slave Modbus code
```iecst
(********************************************************************
 * COPYRIGHT -- Bernecker + Rainer
 ********************************************************************
 * Program: Slave_mbus
 * File: Slave_mbus.st
 * Author: gimeneza
 * Created: March 07, 2017
 ********************************************************************
 * Implementation of program Slave_mbus
 ********************************************************************)

PROGRAM _INIT
	ident := 1;
	(* Create a Modbus server with unit identity = 1, Coil = 0, HoldingRegister = 9000, DiscreteInputs = 0, InputRegister = 0 *)
	BRSE_MB_Alloc(ident,1000,9000,0,0);

	(* Bind the holding registers *)
	FOR i:=0 TO 8999 DO
		BRSE_MB_HoldingRegister(ident,i,ADR(HoldingRegister[i]));
	END_FOR;

END_PROGRAM

PROGRAM _CYCLIC

    (* Enable the server, use INTEL alignment (little endian) for real Values *)
	FB_BRSE_MBT_Server(Enable := 1, ClientFormat := BRSE_MB_INTEL, Port := 502, SocketTimeout:=5000);

END_PROGRAM

PROGRAM _EXIT

    (* Close the open tcp port *)
	FB_MBT_ServerExit();

END_PROGRAM
```

### Package Logical/ExtPack/_Comms/ModbusComms/ModbusComms_v1/Libraries - Modbus libraries

### Library Logical/ExtPack/_Comms/ModbusComms/ModbusComms_v1/Libraries/BRSE_MB (ANSIC, version 1.16.0)
Depends on: AsString, sys_lib, AsIecCon, brsystem

#### BRSE_MB.typ - Exported data types
```iecst
TYPE
	BRSE_MB_ServerUnit_typ : 	STRUCT
		pDiscreteInputs : UDINT; (*address to array of variable addresses, dynamically allocated*)
		pCoils : UDINT;
		pInputRegisters : UDINT;
		pHoldingRegisters : UDINT;
		MaxCoils : UINT; (*(Sizes need to be saved for error handling purposes)*)
		MaxHoldingRegisters : UINT;
		MaxDiscreteInputs : UINT;
		MaxInputRegisters : UINT;
	END_STRUCT;
	BRSE_MB_ServerCfg_typ : 	STRUCT
		Unit : ARRAY[0..255] OF BRSE_MB_ServerUnit_typ;
	END_STRUCT;
	BRSE_MB_Request_typ : 	STRUCT
		Unit : USINT; (*Unit in server*)
		Type : USINT; (*Modbus function code*)
		StartAddr : UINT; (*Reference, where to begin reading/writing*)
		Quantity : UINT; (*Number of items to be read/written*)
	END_STRUCT;
	MB_ClientStruct_typ : 	STRUCT
		pClients : ARRAY[0..255] OF UDINT; (*Clients[ClientID] holds the address to an instance of MB_Client_typ (i.e. the request queue) of that ClientID*)
	END_STRUCT;
	MB_ClientQueueItem_typ : 	STRUCT
		Request : BRSE_MB_Request_typ;
		VariableAddr : UDINT; (*Address where to begin reading/writing variables*)
		StatusAddr : UDINT; (*Address of the status register, where to tell when request has been executed and/or error code.*)
	END_STRUCT;
	MB_Client_typ : 	STRUCT
		Queue : ARRAY[0..MB_QUEUE_SIZE] OF MB_ClientQueueItem_typ;
		IndexExec : UINT; (*Next request in queue to be executed*)
		IndexInsert : UINT; (*Where to insert the next queued request*)
		Lock : BOOL;
	END_STRUCT;
END_TYPE
```

#### BRSE_MB_Main.h
```c
/*! \file BRSE_MB_Main.h */

/*! \mainpage BRSE_MB

	\section Introduction

	This library is used for setting up a modbus server and a modbus client.
	It contains functions for allocating units and bind registers and coils to variables.

	The Modbus data model has a simple structure that differentiates
	between four basic data types:

	\arg Discrete Inputs (BOOL Read-Only)
	\arg Coils (BOOL Read-Write)
	\arg Input Registers (INT Read-Only)
	\arg Holding Registers (INT Read-Write)

	(The expression "Input" is seen from the Client side).

	\section Server

	The server is represented as a function block for responding to modbus messages, by processing an input buffer
	and create an output buffer. This buffer may then be "framed" for the desired communication protocol.
	The server block is used in BRSE_MBR (rtu) and BRSE_MBT (tcp). These libraries (MBT, MBR) create the
	connection to a physical interface such as the Ethernet Port or the Serial port.

	\image html y:\Application\Libraries\BRSE_MB\Documentation\BRSE_MB_Server.jpg

	\par Server Side functions

	BRSE_MB_Alloc  - Allocates space for a unit with the specified number of coils, holding registers, discrete inputs
	and input registers.

	BRSE_MB_Coil - Binds a unit coil reference with a boolean variable.

	BRSE_MB_HoldingRegister - Binds a unit holding register reference with an integer variable.

	BRSE_MB_InputRegister - Binds a unit input register reference with an integer variable.

	BRSE_MB_DiscreteInput - Binds a unit discrete input reference with a boolean variable.

	BRSE_MB_4ByteHoldingRegister - Binds a 4 byte variable to 2 holding registers

	BRSE_MB_Server - Responds to modbus messages by creating the output buffer containing the response. It is used by BRSE_MBR
	and BRSE_MBT and is not usually not implemented directly by the user.

	For an example on how to use this library, see BRSE_MBR or BRSE_MBT.

	\section Client

	The client is represented as a function block for creating modbus messages, by generate a request queue buffer
	and listen for response from the server. This buffer may then be "framed" for the desired communication protocol.
	The client block is used in BRSE_MBR (rtu) and BRSE_MBT (tcp). These libraries (MBT, MBR) create the
	connection to a physical interface such as the Ethernet Port or the Serial port.

	\image html y:\Application\Libraries\BRSE_MB\Documentation\BRSE_MB_Client.jpg

	\par Client Side Functions

	MB_AllocClient - Allocates space for a client request queue.

	MB_ReadDiscreteInputs - Read event triggered from a discreate input.

	MB_ReadCoils - Read event triggered from a coil.

	MB_ReadInputRegisters - Read event triggered from a input register.

	MB_ReadHoldingRegisters - Read event triggered from a holding register.

	MB_PollDiscreteInputs - Read cyclic from a discreate input.

	MB_PollCoils - Read cyclic from a coil.

	MB_PollInputRegisters - Read cyclic from a input register.

	MB_PollHoldingRegisters - Read cyclic from a holding register.

	MB_WriteCoils - Write event triggered to a coil.

	MB_WriteHoldingRegisters - Write event triggered to a holding register.

	MB_PushCoils - Write cyclic to a coil.

	MB_PushHoldingRegisters - Write cyclic to a holding register.

	MB_Poll4ByteHoldingRegisters - Read cyclic from a 4 byte register

	MB_Push4ByteHoldingRegisters - Write cyclic to a 4 byte register

	MB_Write4ByteHoldingRegisters - Write event triggered to a 4 byte register

	MB_Read4ByteHoldingRegisters - Read event triggered from a 4 byte register

	\par Internal Functions

	MB_CreateClientRequest - Create request as a modbus message. It is used by BRSE_MBR and BRSE_MBT and is not usually not implemented directly by the user.

	MB_PutClientResponse - Create respons as a modbus message. It is used by BRSE_MBR and BRSE_MBT and is not usually not implemented directly by the user.

	\par Example

	For an example on how to use this library, see BRSE_MBR or BRSE_MBT.

	When reading and writeing many variables it is convenient to use arrays.
	Just set the address to the first element in the array (FB_MB_WriteCoils.VariablesAddress := ADR(startMotor[0]))
	and set the number of element in the array (FB_MB_WriteCoils.Quantity := 3;)
*/

/*! \page Error_Number Error Numbers and Constants

	\section internal_err Internal Error Numbers

	These error numbers can be set on the Status output of the respective BRSE_MB function block.

	\b 20004 MB_ERR_CLIENT_NOT_ALLOCATED: A request was requested from a client which hasn't been allocated

	\b 20005 MB_ERR_BUFFER: Buffer is too small for request or buffer address is 0

	\b 20006 MB_ERR_QUEUE_FULL: The queue is full

	\b 20007 MB_ERR_INTERNAL: Internal error

	\b 20008 MB_ERR_PROTOCOL: Error in protocol

	\b 20009 MB_ERR_QUANTITY: The quantity is too big or 0

	\section modbus_err Modbus Error Numbers

	These error numbers can be set on the Status output of the respective BRSE_MB function block.

	\b 1 ERROR_ILLEGAL_FUNCTlON
	The function code received in the query is not an allowable action for the slave. This may be
	because the function code is only applicable to newer controllers, and was not implemented in the
	unit selected. It could also indicate that the slave is in the wrong state to process a request of this
	type, for example because it is unconfigured and is being asked to return register values.

	\b 2 ERROR_ILLEGAL_DATA_ADDRESS
	The data address received in the query is not an allowable address for the slave. More specifically,
	the combination of reference number and transfer length is invalid. For a controller with 100
	registers, a request with offset 96 and length 4 would succeed, a request with offset 96 and length
	5 will generate exception 02.

	\b 3 ERROR_ILLEGAL_DATA_VALUE
	A value contained in the query data field is not an allowable value for the slave. This indicates a
	fault in the structure of the remainder of a complex request, such as that the implied length is
	incorrect. It specifically does NOT mean that a data item submitted for storage in a register has a
	value outside the expectation of the application program, since the MODBUS protocol is unaware
	of the significance of any particular value of any particular register.

	\b 4 ERROR_ILLEGAL_RESPONSE_LENGTH
	Indicates that the request as framed would generate a response whose size exceeds the available
	MODBUS data size. Used only by functions generating a multi-part response, such as functions 20 and 21

	\section consts Constants

	These Constants are set to the ServerFormat or ClientFormat inputs to define which Byte-alignment
	that is in use on the opposite station.

	\b 0 	BRSE_MB_INTEL: The server/client on the other side uses the Intel format

	\b 1 	BRSE_MB_MOTOROLA: The server/client on the other side uses the Motorola format

*/

#ifndef _BRSE_MB_MAIN_
#define _BRSE_MB_MAIN_

#include <bur/plctypes.h>
#include "BRSE_MB.h"
#include <string.h>
#include <AsIecCon.h>
#endif

/* internal functions in library */

/* implemented in BRSE_MB_Server.c */
UINT BRSE_MB_ReadCoils(struct BRSE_MB_Server* inst);
UINT BRSE_MB_ReadDiscreteInputs(struct BRSE_MB_Server* inst);
UINT BRSE_MB_ReadHoldingRegisters(struct BRSE_MB_Server* inst);
UINT BRSE_MB_ReadInputRegisters(struct BRSE_MB_Server* inst);
UINT BRSE_MB_WriteSingleCoil(struct BRSE_MB_Server* inst);
UINT BRSE_MB_WriteSingleRegister(struct BRSE_MB_Server* inst);
UINT BRSE_MB_WriteMultipleCoils(struct BRSE_MB_Server* inst);
UINT BRSE_MB_WriteMultipleRegisters(struct BRSE_MB_Server* inst);
UINT BRSE_MB_FillDigitalBuffer(struct BRSE_MB_Server* inst, UDINT *boolPtrArray);
UINT BRSE_MB_FillRegisterBuffer(struct BRSE_MB_Server* inst, UDINT *intPtrArray);

UINT BRSE_MB_FillRegisterBuffer4Byte(USINT ServerFormat, struct BRSE_MB_Server* inst, UDINT *intPtrArray);
void MB_FillRegisterValues4Byte(USINT ServerFormat, USINT *pByteBuffer, MB_ClientQueueItem_typ *pQueueItem);

/* implemented in BRSE_MB_Client.c */
void MB_FillRegisterValues(USINT *pByteBuffer, MB_ClientQueueItem_typ *pQueueItem); /* implemented in this file */
void MB_FillCoilValues(USINT *pByteBuffer, MB_ClientQueueItem_typ *pQueueItem);

/* implemented in MB_RequestQueue.c*/
UINT MB_AddToRequestQueue(USINT clientID, USINT fc, UINT quantity, UINT startAddress, UDINT variableAddress, UDINT statusAddress, USINT Unit);
/* Checking if the queue is presumably alive or dead. 0=dead, 1=alive */
USINT MB_QueueStatus(USINT ClientID);
```
